  MoveL 7456 to (240.92, 51.59, 106.87) mm, rotated rx 180 ry 0 rz 180 deg; joints [-19.251, 9.742, 68.195, 59.104, 22.596, -57.051]
  Call Extruder(211.45578)
  MoveL 7457 to (240.97, 51.98, 106.87) mm, rotated rx -180 ry 0 rz 180 deg; joints [-19.29, 9.772, 68.161, 59.149, 22.631, -57.091]
  MoveL 7458 to (240.97, 51.98, 106.87) mm, rotated rx -180 ry 0 rz 180 deg; joints [-19.29, 9.772, 68.161, 59.149, 22.631, -57.091]
  Call Extruder(211.65249)
  MoveL 7459 to (241.02, 52.37, 106.87) mm, rotated rx 180 ry 0 rz 180 deg; joints [-19.329, 9.801, 68.126, 59.194, 22.666, -57.131]
  MoveL 7460 to (241.02, 52.37, 106.87) mm, rotated rx 180 ry 0 rz 180 deg; joints [-19.329, 9.801, 68.126, 59.194, 22.666, -57.131]
  Call Extruder(211.84833)
  MoveL 7461 to (241.06, 52.75, 106.87) mm, rotated rx 180 ry 0 rz 180 deg; joints [-19.368, 9.831, 68.092, 59.239, 22.702, -57.171]
  MoveL 7462 to (241.06, 52.75, 106.87) mm, rotated rx 180 ry 0 rz 180 deg; joints [-19.368, 9.831, 68.092, 59.239, 22.702, -57.171]
  Call Extruder(212.14376)
  MoveL 7463 to (241.11, 53.34, 106.87) mm, rotated rx -180 ry 0 rz 180 deg; joints [-19.428, 9.872, 68.043, 59.309, 22.756, -57.233]
  MoveL 7464 to (241.11, 53.34, 106.87) mm, rotated rx -180 ry 0 rz 180 deg; joints [-19.428, 9.872, 68.043, 59.309, 22.756, -57.233]
  Call Extruder(212.43787)
  MoveL 7465 to (241.16, 53.93, 106.87) mm, rotated rx 180 ry 0 rz 180 deg; joints [-19.488, 9.914, 67.995, 59.379, 22.81, -57.295]
  MoveL 7466 to (241.16, 53.93, 106.87) mm, rotated rx 180 ry 0 rz 180 deg; joints [-19.488, 9.914, 67.995, 59.379, 22.81, -57.295]
  Call Extruder(212.73064)
  MoveL 7467 to (241.2, 54.52, 106.87) mm, rotated rx 180 ry 0 rz 180 deg; joints [-19.548, 9.956, 67.946, 59.448, 22.864, -57.357]
  MoveL 7468 to (241.2, 54.52, 106.87) mm, rotated rx 180 ry 0 rz 180 deg; joints [-19.548, 9.956, 67.946, 59.448, 22.864, -57.357]
  Call Extruder(213.30409)
  MoveL 7469 to (241.25, 55.68, 106.87) mm, rotated rx 180 ry 0 rz 180 deg; joints [-19.668, 10.031, 67.858, 59.588, 22.971, -57.482]
  MoveL 7470 to (241.25, 55.68, 106.87) mm, rotated rx 180 ry 0 rz 180 deg; joints [-19.668, 10.031, 67.858, 59.588, 22.971, -57.482]
  Call Extruder(214.01793)
  MoveL 7471 to (241.29, 57.14, 106.87) mm, rotated rx 180 ry 0 rz 180 deg; joints [-19.819, 10.123, 67.751, 59.763, 23.106, -57.637]
  Call Extruder(256.08281)
  MoveL 7472 to (241.29, 142.86, 106.87) mm, rotated rx -180 ry 0 rz 180 deg; joints [-28.232, 16.484, 59.966, 66.424, 31.073, -63.002]
  Call Extruder(256.51124)
  MoveL 7473 to (241.27, 143.73, 106.87) mm, rotated rx 180 ry 0 rz -180 deg; joints [-28.313, 16.56, 59.868, 66.463, 31.153, -63.025]
  MoveL 7474 to (241.27, 143.73, 106.87) mm, rotated rx 180 ry 0 rz -180 deg; joints [-28.313, 16.56, 59.868, 66.463, 31.153, -63.025]
  Call Extruder(257.08469)
  MoveL 7475 to (241.22, 144.9, 106.87) mm, rotated rx 180 ry 0 rz 180 deg; joints [-28.421, 16.658, 59.742, 66.516, 31.261, -63.057]
  MoveL 7476 to (241.22, 144.9, 106.87) mm, rotated rx 180 ry 0 rz 180 deg; joints [-28.421, 16.658, 59.742, 66.516, 31.261, -63.057]
  Call Extruder(257.51903)
  MoveL 7477 to (241.18, 145.77, 106.87) mm, rotated rx -180 ry 0 rz 180 deg; joints [-28.503, 16.731, 59.649, 66.557, 31.342, -63.082]
  MoveL 7478 to (241.18, 145.77, 106.87) mm, rotated rx -180 ry 0 rz 180 deg; joints [-28.503, 16.731, 59.649, 66.557, 31.342, -63.082]
  Call Extruder(257.81314)
  MoveL 7479 to (241.13, 146.36, 106.87) mm, rotated rx 180 ry 0 rz 180 deg; joints [-28.559, 16.777, 59.59, 66.586, 31.397, -63.101]
  MoveL 7480 to (241.13, 146.36, 106.87) mm, rotated rx 180 ry 0 rz 180 deg; joints [-28.559, 16.777, 59.59, 66.586, 31.397, -63.101]
  Call Extruder(258.10858)
  MoveL 7481 to (241.09, 146.95, 106.87) mm, rotated rx 180 ry 0 rz 180 deg; joints [-28.615, 16.824, 59.53, 66.615, 31.452, -63.119]
  MoveL 7482 to (241.09, 146.95, 106.87) mm, rotated rx 180 ry 0 rz 180 deg; joints [-28.615, 16.824, 59.53, 66.615, 31.452, -63.119]
  Call Extruder(258.35483)
  MoveL 7483 to (241.04, 147.44, 106.87) mm, rotated rx -180 ry 0 rz 180 deg; joints [-28.662, 16.861, 59.482, 66.639, 31.498, -63.135]
  MoveL 7484 to (241.04, 147.44, 106.87) mm, rotated rx -180 ry 0 rz 180 deg; joints [-28.662, 16.861, 59.482, 66.639, 31.498, -63.135]
  Call Extruder(258.55154)
  MoveL 7485 to (240.99, 147.83, 106.87) mm, rotated rx -180 ry 0 rz 180 deg; joints [-28.7, 16.889, 59.446, 66.66, 31.535, -63.148]
  MoveL 7486 to (240.99, 147.83, 106.87) mm, rotated rx -180 ry 0 rz 180 deg; joints [-28.7, 16.889, 59.446, 66.66, 31.535, -63.148]
  Call Extruder(258.74911)
  MoveL 7487 to (240.95, 148.22, 106.87) mm, rotated rx 180 ry 0 rz 180 deg; joints [-28.737, 16.917, 59.41, 66.68, 31.571, -63.162]
  MoveL 7488 to (240.95, 148.22, 106.87) mm, rotated rx 180 ry 0 rz 180 deg; joints [-28.737, 16.917, 59.41, 66.68, 31.571, -63.162]
  Call Extruder(258.94755)
  MoveL 7489 to (240.9, 148.6, 106.87) mm, rotated rx 180 ry 0 rz 180 deg; joints [-28.774, 16.945, 59.374, 66.7, 31.608, -63.175]
  MoveL 7490 to (240.9, 148.6, 106.87) mm, rotated rx 180 ry 0 rz 180 deg; joints [-28.774, 16.945, 59.374, 66.7, 31.608, -63.175]
  Call Extruder(259.14686)
  MoveL 7491 to (240.86, 148.99, 106.87) mm, rotated rx 180 ry 0 rz 180 deg; joints [-28.812, 16.974, 59.338, 66.72, 31.645, -63.188]
  MoveL 7492 to (240.86, 148.99, 106.87) mm, rotated rx 180 ry 0 rz 180 deg; joints [-28.812, 16.974, 59.338, 66.72, 31.645, -63.188]
  Call Extruder(259.30569)
  MoveL 7493 to (240.81, 149.3, 106.87) mm, rotated rx 180 ry 0 rz 180 deg; joints [-28.842, 16.994, 59.311, 66.737, 31.674, -63.2]
  MoveL 7494 to (240.81, 149.3, 106.87) mm, rotated rx 180 ry 0 rz 180 deg; joints [-28.842, 16.994, 59.311, 66.737, 31.674, -63.2]
  Call Extruder(259.46525)
  MoveL 7495 to (240.76, 149.6, 106.87) mm, rotated rx -180 ry 0 rz 180 deg; joints [-28.872, 17.014, 59.285, 66.755, 31.703, -63.212]
  MoveL 7496 to (240.76, 149.6, 106.87) mm, rotated rx -180 ry 0 rz 180 deg; joints [-28.872, 17.014, 59.285, 66.755, 31.703, -63.212]
  Call Extruder(259.62554)
  MoveL 7497 to (240.71, 149.91, 106.87) mm, rotated rx 180 ry 0 rz 180 deg; joints [-28.902, 17.035, 59.259, 66.772, 31.732, -63.224]
  MoveL 7498 to (240.71, 149.91, 106.87) mm, rotated rx 180 ry 0 rz 180 deg; joints [-28.902, 17.035, 59.259, 66.772, 31.732, -63.224]
  Call Extruder(259.78655)
  MoveL 7499 to (240.66, 150.21, 106.87) mm, rotated rx -180 ry 0 rz -180 deg; joints [-28.932, 17.055, 59.233, 66.789, 31.761, -63.236]
  MoveL 7500 to (240.66, 150.21, 106.87) mm, rotated rx -180 ry 0 rz -180 deg; joints [-28.932, 17.055, 59.233, 66.789, 31.761, -63.236]
  Call Extruder(259.94830)
  MoveL 7501 to (240.61, 150.52, 106.87) mm, rotated rx 180 ry 0 rz 180 deg; joints [-28.962, 17.075, 59.207, 66.806, 31.791, -63.247]
  MoveL 7502 to (240.61, 150.52, 106.87) mm, rotated rx 180 ry 0 rz 180 deg; joints [-28.962, 17.075, 59.207, 66.806, 31.791, -63.247]
  Call Extruder(260.11077)
  MoveL 7503 to (240.57, 150.83, 106.87) mm, rotated rx -180 ry 0 rz 180 deg; joints [-28.993, 17.096, 59.18, 66.823, 31.82, -63.259]
  MoveL 7504 to (240.57, 150.83, 106.87) mm, rotated rx -180 ry 0 rz 180 deg; joints [-28.993, 17.096, 59.18, 66.823, 31.82, -63.259]
  Call Extruder(260.24469)
  MoveL 7505 to (240.52, 151.08, 106.87) mm, rotated rx 180 ry 0 rz 180 deg; joints [-29.017, 17.111, 59.161, 66.838, 31.844, -63.269]
  MoveL 7506 to (240.52, 151.08, 106.87) mm, rotated rx 180 ry 0 rz 180 deg; joints [-29.017, 17.111, 59.161, 66.838, 31.844, -63.269]
  Call Extruder(260.37923)
  MoveL 7507 to (240.47, 151.32, 106.87) mm, rotated rx -180 ry 0 rz 180 deg; joints [-29.043, 17.126, 59.142, 66.853, 31.868, -63.28]
  MoveL 7508 to (240.47, 151.32, 106.87) mm, rotated rx -180 ry 0 rz 180 deg; joints [-29.043, 17.126, 59.142, 66.853, 31.868, -63.28]
  Call Extruder(260.51438)
  MoveL 7509 to (240.42, 151.57, 106.87) mm, rotated rx 180 ry 0 rz 180 deg; joints [-29.067, 17.141, 59.122, 66.868, 31.892, -63.29]
  MoveL 7510 to (240.42, 151.57, 106.87) mm, rotated rx 180 ry 0 rz 180 deg; joints [-29.067, 17.141, 59.122, 66.868, 31.892, -63.29]
  Call Extruder(260.65014)
  MoveL 7511 to (240.37, 151.82, 106.87) mm, rotated rx -180 ry 0 rz 180 deg; joints [-29.092, 17.156, 59.103, 66.882, 31.916, -63.301]
  MoveL 7512 to (240.37, 151.82, 106.87) mm, rotated rx -180 ry 0 rz 180 deg; joints [-29.092, 17.156, 59.103, 66.882, 31.916, -63.301]
  Call Extruder(260.78650)
  MoveL 7513 to (240.32, 152.07, 106.87) mm, rotated rx 180 ry 0 rz 180 deg; joints [-29.117, 17.171, 59.083, 66.897, 31.94, -63.311]
  MoveL 7514 to (240.32, 152.07, 106.87) mm, rotated rx 180 ry 0 rz 180 deg; joints [-29.117, 17.171, 59.083, 66.897, 31.94, -63.311]
  Call Extruder(260.92348)
  MoveL 7515 to (240.27, 152.32, 106.87) mm, rotated rx -180 ry 0 rz 180 deg; joints [-29.142, 17.186, 59.064, 66.912, 31.964, -63.321]
  MoveL 7516 to (240.27, 152.32, 106.87) mm, rotated rx -180 ry 0 rz 180 deg; joints [-29.142, 17.186, 59.064, 66.912, 31.964, -63.321]
  Call Extruder(261.06107)
  MoveL 7517 to (240.22, 152.57, 106.87) mm, rotated rx -180 ry 0 rz 180 deg; joints [-29.167, 17.201, 59.044, 66.926, 31.988, -63.332]
  MoveL 7518 to (240.22, 152.57, 106.87) mm, rotated rx -180 ry 0 rz 180 deg; joints [-29.167, 17.201, 59.044, 66.926, 31.988, -63.332]
  Call Extruder(261.17477)
  MoveL 7519 to (240.17, 152.77, 106.87) mm, rotated rx 180 ry 0 rz 180 deg; joints [-29.188, 17.213, 59.029, 66.939, 32.008, -63.341]
  MoveL 7520 to (240.17, 152.77, 106.87) mm, rotated rx 180 ry 0 rz 180 deg; joints [-29.188, 17.213, 59.029, 66.939, 32.008, -63.341]
  Call Extruder(261.28892)
  MoveL 7521 to (240.13, 152.98, 106.87) mm, rotated rx 180 ry 0 rz 180 deg; joints [-29.209, 17.225, 59.014, 66.951, 32.027, -63.35]
  MoveL 7522 to (240.13, 152.98, 106.87) mm, rotated rx 180 ry 0 rz 180 deg; joints [-29.209, 17.225, 59.014, 66.951, 32.027, -63.35]
  Call Extruder(261.40352)
  MoveL 7523 to (240.08, 153.18, 106.87) mm, rotated rx 180 ry 0 rz 180 deg; joints [-29.229, 17.237, 58.999, 66.964, 32.047, -63.358]
  MoveL 7524 to (240.08, 153.18, 106.87) mm, rotated rx 180 ry 0 rz 180 deg; joints [-29.229, 17.237, 58.999, 66.964, 32.047, -63.358]
  Call Extruder(261.51858)
  MoveL 7525 to (240.04, 153.39, 106.87) mm, rotated rx 180 ry 0 rz 180 deg; joints [-29.25, 17.248, 58.983, 66.976, 32.067, -63.367]
  MoveL 7526 to (240.04, 153.39, 106.87) mm, rotated rx 180 ry 0 rz 180 deg; joints [-29.25, 17.248, 58.983, 66.976, 32.067, -63.367]
  Call Extruder(261.64080)
  MoveL 7527 to (239.98, 153.6, 106.87) mm, rotated rx 180 ry 0 rz 180 deg; joints [-29.272, 17.259, 58.97, 66.99, 32.088, -63.378]
  MoveL 7528 to (239.98, 153.6, 106.87) mm, rotated rx 180 ry 0 rz 180 deg; joints [-29.272, 17.259, 58.97, 66.99, 32.088, -63.378]
  Call Extruder(261.77046)
  MoveL 7529 to (239.92, 153.82, 106.87) mm, rotated rx -180 ry 0 rz 180 deg; joints [-29.296, 17.269, 58.957, 67.006, 32.11, -63.389]
  MoveL 7530 to (239.92, 153.82, 106.87) mm, rotated rx -180 ry 0 rz 180 deg; joints [-29.296, 17.269, 58.957, 67.006, 32.11, -63.389]
  Call Extruder(261.90069)
  MoveL 7531 to (239.85, 154.05, 106.87) mm, rotated rx 180 ry 0 rz 180 deg; joints [-29.319, 17.279, 58.944, 67.021, 32.132, -63.401]
  MoveL 7532 to (239.85, 154.05, 106.87) mm, rotated rx 180 ry 0 rz 180 deg; joints [-29.319, 17.279, 58.944, 67.021, 32.132, -63.401]
  Call Extruder(262.03148)
  MoveL 7533 to (239.78, 154.27, 106.87) mm, rotated rx 180 ry 0 rz 180 deg; joints [-29.343, 17.289, 58.932, 67.037, 32.155, -63.413]
  MoveL 7534 to (239.78, 154.27, 106.87) mm, rotated rx 180 ry 0 rz 180 deg; joints [-29.343, 17.289, 58.932, 67.037, 32.155, -63.413]
  Call Extruder(262.16284)
  MoveL 7535 to (239.71, 154.5, 106.87) mm, rotated rx 180 ry 0 rz -180 deg; joints [-29.366, 17.299, 58.919, 67.053, 32.177, -63.425]
  MoveL 7536 to (239.71, 154.5, 106.87) mm, rotated rx 180 ry 0 rz -180 deg; joints [-29.366, 17.299, 58.919, 67.053, 32.177, -63.425]
  Call Extruder(262.27474)
  MoveL 7537 to (239.65, 154.68, 106.87) mm, rotated rx 180 ry 0 rz 180 deg; joints [-29.386, 17.306, 58.909, 67.066, 32.195, -63.435]
  MoveL 7538 to (239.65, 154.68, 106.87) mm, rotated rx 180 ry 0 rz 180 deg; joints [-29.386, 17.306, 58.909, 67.066, 32.195, -63.435]
  Call Extruder(262.38708)
  MoveL 7539 to (239.59, 154.87, 106.87) mm, rotated rx 180 ry 0 rz -180 deg; joints [-29.406, 17.314, 58.899, 67.08, 32.214, -63.446]
  MoveL 7540 to (239.59, 154.87, 106.87) mm, rotated rx 180 ry 0 rz -180 deg; joints [-29.406, 17.314, 58.899, 67.08, 32.214, -63.446]
  Call Extruder(262.49987)
  MoveL 7541 to (239.53, 155.06, 106.87) mm, rotated rx 180 ry 0 rz 180 deg; joints [-29.426, 17.321, 58.889, 67.093, 32.233, -63.456]
  MoveL 7542 to (239.53, 155.06, 106.87) mm, rotated rx 180 ry 0 rz 180 deg; joints [-29.426, 17.321, 58.889, 67.093, 32.233, -63.456]
  Call Extruder(262.61311)
  MoveL 7543 to (239.47, 155.25, 106.87) mm, rotated rx 180 ry 0 rz 180 deg; joints [-29.446, 17.329, 58.879, 67.107, 32.252, -63.466]
  MoveL 7544 to (239.47, 155.25, 106.87) mm, rotated rx 180 ry 0 rz 180 deg; joints [-29.446, 17.329, 58.879, 67.107, 32.252, -63.466]
  Call Extruder(262.72679)
  MoveL 7545 to (239.41, 155.44, 106.87) mm, rotated rx 180 ry 0 rz 180 deg; joints [-29.466, 17.337, 58.87, 67.12, 32.271, -63.477]
  MoveL 7546 to (239.41, 155.44, 106.87) mm, rotated rx 180 ry 0 rz 180 deg; joints [-29.466, 17.337, 58.87, 67.12, 32.271, -63.477]
  Call Extruder(262.90875)
  MoveL 7547 to (239.29, 155.73, 106.87) mm, rotated rx -180 ry 0 rz 180 deg; joints [-29.499, 17.344, 58.86, 67.144, 32.3, -63.496]
  MoveL 7548 to (239.29, 155.73, 106.87) mm, rotated rx -180 ry 0 rz 180 deg; joints [-29.499, 17.344, 58.86, 67.144, 32.3, -63.496]
  Call Extruder(263.09146)
  MoveL 7549 to (239.17, 156.02, 106.87) mm, rotated rx 180 ry 0 rz 180 deg; joints [-29.531, 17.352, 58.85, 67.168, 32.33, -63.515]
  MoveL 7550 to (239.17, 156.02, 106.87) mm, rotated rx 180 ry 0 rz 180 deg; joints [-29.531, 17.352, 58.85, 67.168, 32.33, -63.515]
  Call Extruder(263.26189)
  MoveL 7551 to (239.05, 156.29, 106.87) mm, rotated rx 180 ry 0 rz 180 deg; joints [-29.561, 17.358, 58.842, 67.19, 32.358, -63.533]
  MoveL 7552 to (239.05, 156.29, 106.87) mm, rotated rx 180 ry 0 rz 180 deg; joints [-29.561, 17.358, 58.842, 67.19, 32.358, -63.533]
  Call Extruder(263.41990)
  MoveL 7553 to (238.94, 156.54, 106.87) mm, rotated rx 180 ry 0 rz 180 deg; joints [-29.589, 17.364, 58.834, 67.211, 32.383, -63.549]
  MoveL 7554 to (238.94, 156.54, 106.87) mm, rotated rx 180 ry 0 rz 180 deg; joints [-29.589, 17.364, 58.834, 67.211, 32.383, -63.549]
  Call Extruder(263.57851)
  MoveL 7555 to (238.84, 156.79, 106.87) mm, rotated rx 180 ry 0 rz 180 deg; joints [-29.617, 17.37, 58.827, 67.231, 32.409, -63.566]
  MoveL 7556 to (238.84, 156.79, 106.87) mm, rotated rx 180 ry 0 rz 180 deg; joints [-29.617, 17.37, 58.827, 67.231, 32.409, -63.566]
  Call Extruder(263.78468)
  MoveL 7557 to (238.66, 157.09, 106.87) mm, rotated rx 180 ry 0 rz 180 deg; joints [-29.653, 17.37, 58.827, 67.262, 32.441, -63.591]
  MoveL 7558 to (238.66, 157.09, 106.87) mm, rotated rx 180 ry 0 rz 180 deg; joints [-29.653, 17.37, 58.827, 67.262, 32.441, -63.591]
  Call Extruder(263.99163)
  MoveL 7559 to (238.49, 157.4, 106.87) mm, rotated rx 180 ry 0 rz 180 deg; joints [-29.689, 17.369, 58.828, 67.292, 32.474, -63.617]
  MoveL 7560 to (238.49, 157.4, 106.87) mm, rotated rx 180 ry 0 rz 180 deg; joints [-29.689, 17.369, 58.828, 67.292, 32.474, -63.617]
  Call Extruder(264.19935)
  MoveL 7561 to (238.31, 157.7, 106.87) mm, rotated rx 180 ry 0 rz -180 deg; joints [-29.725, 17.369, 58.828, 67.322, 32.506, -63.642]
  MoveL 7562 to (238.31, 157.7, 106.87) mm, rotated rx 180 ry 0 rz -180 deg; joints [-29.725, 17.369, 58.828, 67.322, 32.506, -63.642]
  Call Extruder(264.40786)
  MoveL 7563 to (238.13, 158.01, 106.87) mm, rotated rx 180 ry 0 rz 180 deg; joints [-29.761, 17.368, 58.828, 67.352, 32.538, -63.668]
  MoveL 7564 to (238.13, 158.01, 106.87) mm, rotated rx 180 ry 0 rz 180 deg; joints [-29.761, 17.368, 58.828, 67.352, 32.538, -63.668]
  Call Extruder(264.58740)
  MoveL 7565 to (237.96, 158.25, 106.87) mm, rotated rx 180 ry 0 rz 180 deg; joints [-29.792, 17.362, 58.836, 67.38, 32.566, -63.692]
  MoveL 7566 to (237.96, 158.25, 106.87) mm, rotated rx 180 ry 0 rz 180 deg; joints [-29.792, 17.362, 58.836, 67.38, 32.566, -63.692]
  Call Extruder(264.92080)
  MoveL 7567 to (237.63, 158.7, 106.87) mm, rotated rx 180 ry 0 rz 180 deg; joints [-29.849, 17.351, 58.851, 67.432, 32.615, -63.738]
  MoveL 7568 to (237.63, 158.7, 106.87) mm, rotated rx 180 ry 0 rz 180 deg; joints [-29.849, 17.351, 58.851, 67.432, 32.615, -63.738]
  Call Extruder(265.25540)
  MoveL 7569 to (237.3, 159.15, 106.87) mm, rotated rx -180 ry 0 rz 180 deg; joints [-29.907, 17.339, 58.866, 67.484, 32.666, -63.783]
  Call Extruder(266.08335)
  MoveL 7570 to (236.39, 160.19, 106.87) mm, rotated rx 180 ry 0 rz 180 deg; joints [-30.046, 17.286, 58.935, 67.62, 32.785, -63.905]
  Call Extruder(266.91129)
  MoveL 7571 to (235.35, 161.1, 106.87) mm, rotated rx 180 ry 0 rz 180 deg; joints [-30.182, 17.201, 59.045, 67.765, 32.897, -64.039]
  Call Extruder(267.07860)
  MoveL 7572 to (235.13, 161.27, 106.87) mm, rotated rx 180 ry 0 rz 180 deg; joints [-30.208, 17.179, 59.073, 67.795, 32.918, -64.068]
  MoveL 7573 to (235.13, 161.27, 106.87) mm, rotated rx 180 ry 0 rz 180 deg; joints [-30.208, 17.179, 59.073, 67.795, 32.918, -64.068]
  Call Extruder(267.41202)
  MoveL 7574 to (234.68, 161.6, 106.87) mm, rotated rx 180 ry 0 rz 180 deg; joints [-30.261, 17.136, 59.129, 67.855, 32.961, -64.125]
  MoveL 7575 to (234.68, 161.6, 106.87) mm, rotated rx 180 ry 0 rz 180 deg; joints [-30.261, 17.136, 59.129, 67.855, 32.961, -64.125]
  Call Extruder(267.74426)
  MoveL 7576 to (234.23, 161.92, 106.87) mm, rotated rx 180 ry 0 rz 180 deg; joints [-30.314, 17.092, 59.185, 67.916, 33.004, -64.182]
  MoveL 7577 to (234.23, 161.92, 106.87) mm, rotated rx 180 ry 0 rz 180 deg; joints [-30.314, 17.092, 59.185, 67.916, 33.004, -64.182]
  Call Extruder(267.86192)
  MoveL 7578 to (234.05, 162.02, 106.87) mm, rotated rx 180 ry 0 rz -180 deg; joints [-30.331, 17.073, 59.209, 67.938, 33.018, -64.203]
  MoveL 7579 to (234.05, 162.02, 106.87) mm, rotated rx 180 ry 0 rz -180 deg; joints [-30.331, 17.073, 59.209, 67.938, 33.018, -64.203]
  Call Extruder(268.06964)
  MoveL 7580 to (233.75, 162.2, 106.87) mm, rotated rx 180 ry 0 rz 180 deg; joints [-30.363, 17.04, 59.253, 67.977, 33.043, -64.24]
  MoveL 7581 to (233.75, 162.2, 106.87) mm, rotated rx 180 ry 0 rz 180 deg; joints [-30.363, 17.04, 59.253, 67.977, 33.043, -64.24]
  Call Extruder(268.27659)
  MoveL 7582 to (233.45, 162.37, 106.87) mm, rotated rx 180 ry 0 rz 180 deg; joints [-30.394, 17.006, 59.296, 68.015, 33.067, -64.278]
  MoveL 7583 to (233.45, 162.37, 106.87) mm, rotated rx 180 ry 0 rz 180 deg; joints [-30.394, 17.006, 59.296, 68.015, 33.067, -64.278]
  Call Extruder(268.48276)
  MoveL 7584 to (233.14, 162.55, 106.87) mm, rotated rx -180 ry 0 rz -180 deg; joints [-30.426, 16.973, 59.339, 68.054, 33.092, -64.315]
  MoveL 7585 to (233.14, 162.55, 106.87) mm, rotated rx -180 ry 0 rz -180 deg; joints [-30.426, 16.973, 59.339, 68.054, 33.092, -64.315]
  Call Extruder(268.66443)
  MoveL 7586 to (232.87, 162.69, 106.87) mm, rotated rx 180 ry 0 rz 180 deg; joints [-30.453, 16.94, 59.38, 68.089, 33.113, -64.349]
  MoveL 7587 to (232.87, 162.69, 106.87) mm, rotated rx 180 ry 0 rz 180 deg; joints [-30.453, 16.94, 59.38, 68.089, 33.113, -64.349]
  Call Extruder(268.82240)
  MoveL 7588 to (232.62, 162.8, 106.87) mm, rotated rx 180 ry 0 rz 180 deg; joints [-30.476, 16.909, 59.42, 68.119, 33.13, -64.379]
  MoveL 7589 to (232.62, 162.8, 106.87) mm, rotated rx 180 ry 0 rz 180 deg; joints [-30.476, 16.909, 59.42, 68.119, 33.13, -64.379]
  Call Extruder(268.97977)
  MoveL 7590 to (232.37, 162.91, 106.87) mm, rotated rx 180 ry 0 rz 180 deg; joints [-30.498, 16.878, 59.46, 68.15, 33.147, -64.409]
  MoveL 7591 to (232.37, 162.91, 106.87) mm, rotated rx 180 ry 0 rz 180 deg; joints [-30.498, 16.878, 59.46, 68.15, 33.147, -64.409]
  Call Extruder(269.16252)
  MoveL 7592 to (232.08, 163.03, 106.87) mm, rotated rx 180 ry 0 rz 180 deg; joints [-30.524, 16.842, 59.507, 68.185, 33.167, -64.444]
  MoveL 7593 to (232.08, 163.03, 106.87) mm, rotated rx 180 ry 0 rz 180 deg; joints [-30.524, 16.842, 59.507, 68.185, 33.167, -64.444]
  Call Extruder(269.34450)
  MoveL 7594 to (231.78, 163.15, 106.87) mm, rotated rx 180 ry 0 rz -180 deg; joints [-30.551, 16.805, 59.554, 68.22, 33.187, -64.479]
  MoveL 7595 to (231.78, 163.15, 106.87) mm, rotated rx 180 ry 0 rz -180 deg; joints [-30.551, 16.805, 59.554, 68.22, 33.187, -64.479]
  Call Extruder(269.49184)
  MoveL 7596 to (231.54, 163.24, 106.87) mm, rotated rx 180 ry 0 rz 180 deg; joints [-30.571, 16.774, 59.594, 68.249, 33.202, -64.507]
  MoveL 7597 to (231.54, 163.24, 106.87) mm, rotated rx 180 ry 0 rz 180 deg; joints [-30.571, 16.774, 59.594, 68.249, 33.202, -64.507]
  Call Extruder(269.60506)
  MoveL 7598 to (231.35, 163.3, 106.87) mm, rotated rx 180 ry 0 rz 180 deg; joints [-30.587, 16.749, 59.626, 68.271, 33.214, -64.529]
  MoveL 7599 to (231.35, 163.3, 106.87) mm, rotated rx 180 ry 0 rz 180 deg; joints [-30.587, 16.749, 59.626, 68.271, 33.214, -64.529]
  Call Extruder(269.71784)
  MoveL 7600 to (231.17, 163.36, 106.87) mm, rotated rx 180 ry 0 rz 180 deg; joints [-30.602, 16.724, 59.658, 68.294, 33.225, -64.552]
  MoveL 7601 to (231.17, 163.36, 106.87) mm, rotated rx 180 ry 0 rz 180 deg; joints [-30.602, 16.724, 59.658, 68.294, 33.225, -64.552]
  Call Extruder(269.83017)
  MoveL 7602 to (230.98, 163.42, 106.87) mm, rotated rx 180 ry 0 rz 180 deg; joints [-30.618, 16.699, 59.691, 68.316, 33.236, -64.574]
  MoveL 7603 to (230.98, 163.42, 106.87) mm, rotated rx 180 ry 0 rz 180 deg; joints [-30.618, 16.699, 59.691, 68.316, 33.236, -64.574]
  Call Extruder(269.94206)
  MoveL 7604 to (230.79, 163.48, 106.87) mm, rotated rx 180 ry 0 rz 180 deg; joints [-30.633, 16.673, 59.723, 68.338, 33.248, -64.596]
  MoveL 7605 to (230.79, 163.48, 106.87) mm, rotated rx 180 ry 0 rz 180 deg; joints [-30.633, 16.673, 59.723, 68.338, 33.248, -64.596]
  Call Extruder(270.06346)
  MoveL 7606 to (230.58, 163.55, 106.87) mm, rotated rx -180 ry 0 rz 180 deg; joints [-30.65, 16.646, 59.758, 68.362, 33.26, -64.62]
  MoveL 7607 to (230.58, 163.55, 106.87) mm, rotated rx -180 ry 0 rz 180 deg; joints [-30.65, 16.646, 59.758, 68.362, 33.26, -64.62]
  Call Extruder(270.19428)
  MoveL 7608 to (230.36, 163.62, 106.87) mm, rotated rx 180 ry 0 rz 180 deg; joints [-30.668, 16.615, 59.797, 68.388, 33.273, -64.646]
  MoveL 7609 to (230.36, 163.62, 106.87) mm, rotated rx 180 ry 0 rz 180 deg; joints [-30.668, 16.615, 59.797, 68.388, 33.273, -64.646]
  Call Extruder(270.32452)
  MoveL 7610 to (230.14, 163.68, 106.87) mm, rotated rx 180 ry 0 rz 180 deg; joints [-30.685, 16.585, 59.836, 68.414, 33.286, -64.672]
  MoveL 7611 to (230.14, 163.68, 106.87) mm, rotated rx 180 ry 0 rz 180 deg; joints [-30.685, 16.585, 59.836, 68.414, 33.286, -64.672]
  Call Extruder(270.45421)
  MoveL 7612 to (229.91, 163.75, 106.87) mm, rotated rx 180 ry 0 rz 180 deg; joints [-30.703, 16.555, 59.875, 68.44, 33.299, -64.698]
  MoveL 7613 to (229.91, 163.75, 106.87) mm, rotated rx 180 ry 0 rz 180 deg; joints [-30.703, 16.555, 59.875, 68.44, 33.299, -64.698]
  Call Extruder(270.58333)
  MoveL 7614 to (229.69, 163.82, 106.87) mm, rotated rx 180 ry 0 rz 180 deg; joints [-30.721, 16.525, 59.913, 68.466, 33.312, -64.724]
  MoveL 7615 to (229.69, 163.82, 106.87) mm, rotated rx 180 ry 0 rz 180 deg; joints [-30.721, 16.525, 59.913, 68.466, 33.312, -64.724]
  Call Extruder(270.69840)
  MoveL 7616 to (229.48, 163.86, 106.87) mm, rotated rx 180 ry 0 rz 180 deg; joints [-30.736, 16.495, 59.951, 68.489, 33.322, -64.747]
  MoveL 7617 to (229.48, 163.86, 106.87) mm, rotated rx 180 ry 0 rz 180 deg; joints [-30.736, 16.495, 59.951, 68.489, 33.322, -64.747]
  Call Extruder(270.81302)
  MoveL 7618 to (229.28, 163.91, 106.87) mm, rotated rx 180 ry 0 rz 180 deg; joints [-30.751, 16.466, 59.988, 68.512, 33.333, -64.771]
  MoveL 7619 to (229.28, 163.91, 106.87) mm, rotated rx 180 ry 0 rz 180 deg; joints [-30.751, 16.466, 59.988, 68.512, 33.333, -64.771]
  Call Extruder(270.92719)
  MoveL 7620 to (229.08, 163.95, 106.87) mm, rotated rx -180 ry 0 rz -180 deg; joints [-30.766, 16.437, 60.025, 68.535, 33.343, -64.794]
  MoveL 7621 to (229.08, 163.95, 106.87) mm, rotated rx -180 ry 0 rz -180 deg; joints [-30.766, 16.437, 60.025, 68.535, 33.343, -64.794]
  Call Extruder(271.04091)
  MoveL 7622 to (228.87, 164, 106.87) mm, rotated rx 180 ry 0 rz 180 deg; joints [-30.781, 16.408, 60.063, 68.558, 33.354, -64.817]
  MoveL 7623 to (228.87, 164, 106.87) mm, rotated rx 180 ry 0 rz 180 deg; joints [-30.781, 16.408, 60.063, 68.558, 33.354, -64.817]
  Call Extruder(271.16633)
  MoveL 7624 to (228.64, 164.04, 106.87) mm, rotated rx 180 ry 0 rz -180 deg; joints [-30.797, 16.375, 60.104, 68.583, 33.365, -64.843]
  MoveL 7625 to (228.64, 164.04, 106.87) mm, rotated rx 180 ry 0 rz -180 deg; joints [-30.797, 16.375, 60.104, 68.583, 33.365, -64.843]
  Call Extruder(271.30331)
  MoveL 7626 to (228.4, 164.09, 106.87) mm, rotated rx -180 ry 0 rz 180 deg; joints [-30.815, 16.339, 60.15, 68.611, 33.378, -64.871]
  MoveL 7627 to (228.4, 164.09, 106.87) mm, rotated rx -180 ry 0 rz 180 deg; joints [-30.815, 16.339, 60.15, 68.611, 33.378, -64.871]
  Call Extruder(271.43968)
  MoveL 7628 to (228.15, 164.14, 106.87) mm, rotated rx 180 ry 0 rz 180 deg; joints [-30.832, 16.303, 60.196, 68.638, 33.39, -64.9]
  MoveL 7629 to (228.15, 164.14, 106.87) mm, rotated rx 180 ry 0 rz 180 deg; joints [-30.832, 16.303, 60.196, 68.638, 33.39, -64.9]
  Call Extruder(271.57543)
  MoveL 7630 to (227.9, 164.19, 106.87) mm, rotated rx -180 ry 0 rz 180 deg; joints [-30.85, 16.267, 60.242, 68.666, 33.403, -64.928]
  MoveL 7631 to (227.9, 164.19, 106.87) mm, rotated rx -180 ry 0 rz 180 deg; joints [-30.85, 16.267, 60.242, 68.666, 33.403, -64.928]
  Call Extruder(271.71058)
  MoveL 7632 to (227.65, 164.24, 106.87) mm, rotated rx 180 ry 0 rz 180 deg; joints [-30.868, 16.231, 60.288, 68.694, 33.415, -64.956]
  MoveL 7633 to (227.65, 164.24, 106.87) mm, rotated rx 180 ry 0 rz 180 deg; joints [-30.868, 16.231, 60.288, 68.694, 33.415, -64.956]
  Call Extruder(271.84512)
  MoveL 7634 to (227.4, 164.29, 106.87) mm, rotated rx 180 ry 0 rz 180 deg; joints [-30.886, 16.195, 60.333, 68.721, 33.428, -64.984]
  MoveL 7635 to (227.4, 164.29, 106.87) mm, rotated rx 180 ry 0 rz 180 deg; joints [-30.886, 16.195, 60.333, 68.721, 33.428, -64.984]
  Call Extruder(271.97904)
  MoveL 7636 to (227.15, 164.34, 106.87) mm, rotated rx -180 ry 0 rz 180 deg; joints [-30.903, 16.16, 60.379, 68.748, 33.44, -65.012]
  MoveL 7637 to (227.15, 164.34, 106.87) mm, rotated rx -180 ry 0 rz 180 deg; joints [-30.903, 16.16, 60.379, 68.748, 33.44, -65.012]
  Call Extruder(272.12691)
  MoveL 7638 to (226.87, 164.39, 106.87) mm, rotated rx -180 ry 0 rz 180 deg; joints [-30.923, 16.119, 60.431, 68.779, 33.454, -65.042]
  MoveL 7639 to (226.87, 164.39, 106.87) mm, rotated rx -180 ry 0 rz 180 deg; joints [-30.923, 16.119, 60.431, 68.779, 33.454, -65.042]
  Call Extruder(272.28865)
  MoveL 7640 to (226.57, 164.44, 106.87) mm, rotated rx 180 ry 0 rz 180 deg; joints [-30.943, 16.074, 60.488, 68.812, 33.468, -65.076]
  MoveL 7641 to (226.57, 164.44, 106.87) mm, rotated rx 180 ry 0 rz 180 deg; joints [-30.943, 16.074, 60.488, 68.812, 33.468, -65.076]
  Call Extruder(272.44966)
  MoveL 7642 to (226.26, 164.49, 106.87) mm, rotated rx 180 ry 0 rz 180 deg; joints [-30.964, 16.029, 60.545, 68.845, 33.482, -65.11]
  MoveL 7643 to (226.26, 164.49, 106.87) mm, rotated rx 180 ry 0 rz 180 deg; joints [-30.964, 16.029, 60.545, 68.845, 33.482, -65.11]
  Call Extruder(272.60995)
  MoveL 7644 to (225.95, 164.53, 106.87) mm, rotated rx 180 ry 0 rz 180 deg; joints [-30.985, 15.984, 60.602, 68.878, 33.497, -65.144]
  MoveL 7645 to (225.95, 164.53, 106.87) mm, rotated rx 180 ry 0 rz 180 deg; joints [-30.985, 15.984, 60.602, 68.878, 33.497, -65.144]
  Call Extruder(272.76951)
  MoveL 7646 to (225.65, 164.58, 106.87) mm, rotated rx 180 ry 0 rz 180 deg; joints [-31.006, 15.939, 60.659, 68.911, 33.511, -65.178]
  MoveL 7647 to (225.65, 164.58, 106.87) mm, rotated rx 180 ry 0 rz 180 deg; joints [-31.006, 15.939, 60.659, 68.911, 33.511, -65.178]
  Call Extruder(272.92834)
  MoveL 7648 to (225.34, 164.63, 106.87) mm, rotated rx 180 ry 0 rz 180 deg; joints [-31.027, 15.894, 60.716, 68.943, 33.526, -65.211]
  MoveL 7649 to (225.34, 164.63, 106.87) mm, rotated rx 180 ry 0 rz 180 deg; joints [-31.027, 15.894, 60.716, 68.943, 33.526, -65.211]
  Call Extruder(273.10701)
  MoveL 7650 to (225, 164.68, 106.87) mm, rotated rx 180 ry 0 rz -180 deg; joints [-31.049, 15.842, 60.782, 68.98, 33.542, -65.249]
  MoveL 7651 to (225, 164.68, 106.87) mm, rotated rx 180 ry 0 rz -180 deg; joints [-31.049, 15.842, 60.782, 68.98, 33.542, -65.249]
  Call Extruder(273.30545)
  MoveL 7652 to (224.61, 164.72, 106.87) mm, rotated rx -180 ry 0 rz 180 deg; joints [-31.074, 15.784, 60.856, 69.021, 33.559, -65.291]
  MoveL 7653 to (224.61, 164.72, 106.87) mm, rotated rx -180 ry 0 rz 180 deg; joints [-31.074, 15.784, 60.856, 69.021, 33.559, -65.291]
  Call Extruder(273.50302)
  MoveL 7654 to (224.22, 164.77, 106.87) mm, rotated rx -180 ry 0 rz 180 deg; joints [-31.1, 15.726, 60.929, 69.062, 33.576, -65.333]
  MoveL 7655 to (224.22, 164.77, 106.87) mm, rotated rx -180 ry 0 rz 180 deg; joints [-31.1, 15.726, 60.929, 69.062, 33.576, -65.333]
  Call Extruder(273.69973)
  MoveL 7656 to (223.84, 164.82, 106.87) mm, rotated rx -180 ry 0 rz -180 deg; joints [-31.125, 15.668, 61.003, 69.102, 33.594, -65.375]
  MoveL 7657 to (223.84, 164.82, 106.87) mm, rotated rx -180 ry 0 rz -180 deg; joints [-31.125, 15.668, 61.003, 69.102, 33.594, -65.375]
  Call Extruder(273.89557)
  MoveL 7658 to (223.45, 164.86, 106.87) mm, rotated rx -180 ry 0 rz 180 deg; joints [-31.15, 15.61, 61.076, 69.143, 33.611, -65.416]
  MoveL 7659 to (223.45, 164.86, 106.87) mm, rotated rx -180 ry 0 rz 180 deg; joints [-31.15, 15.61, 61.076, 69.143, 33.611, -65.416]
  Call Extruder(274.19092)
  MoveL 7660 to (222.86, 164.91, 106.87) mm, rotated rx 180 ry 0 rz 180 deg; joints [-31.186, 15.519, 61.19, 69.203, 33.635, -65.479]
  MoveL 7661 to (222.86, 164.91, 106.87) mm, rotated rx 180 ry 0 rz 180 deg; joints [-31.186, 15.519, 61.19, 69.203, 33.635, -65.479]
  Call Extruder(274.48494)
  MoveL 7662 to (222.27, 164.96, 106.87) mm, rotated rx -180 ry 0 rz 180 deg; joints [-31.222, 15.429, 61.304, 69.263, 33.66, -65.541]
  MoveL 7663 to (222.27, 164.96, 106.87) mm, rotated rx -180 ry 0 rz 180 deg; joints [-31.222, 15.429, 61.304, 69.263, 33.66, -65.541]
  Call Extruder(274.77764)
  MoveL 7664 to (221.68, 165, 106.87) mm, rotated rx 180 ry 0 rz 180 deg; joints [-31.258, 15.339, 61.418, 69.323, 33.685, -65.603]
  MoveL 7665 to (221.68, 165, 106.87) mm, rotated rx 180 ry 0 rz 180 deg; joints [-31.258, 15.339, 61.418, 69.323, 33.685, -65.603]
  Call Extruder(275.35108)
  MoveL 7666 to (220.52, 165.05, 106.87) mm, rotated rx -180 ry 0 rz 180 deg; joints [-31.326, 15.157, 61.646, 69.439, 33.73, -65.724]
  MoveL 7667 to (220.52, 165.05, 106.87) mm, rotated rx -180 ry 0 rz 180 deg; joints [-31.326, 15.157, 61.646, 69.439, 33.73, -65.724]
  Call Extruder(276.06510)
  MoveL 7668 to (219.06, 165.09, 106.87) mm, rotated rx -180 ry 0 rz 180 deg; joints [-31.409, 14.929, 61.932, 69.581, 33.786, -65.872]
  Call Extruder(392.91185)
  MoveL 7669 to (-19.06, 165.09, 106.87) mm, rotated rx 180 ry 0 rz 180 deg; joints [-51.475, -13.949, 91.048, 79.921, 52.618, -73.682]
  Call Extruder(393.34045)
  MoveL 7670 to (-19.94, 165.07, 106.87) mm, rotated rx -180 ry 0 rz 180 deg; joints [-51.582, -14.03, 91.11, 79.944, 52.723, -73.681]
  MoveL 7671 to (-19.94, 165.07, 106.87) mm, rotated rx -180 ry 0 rz 180 deg; joints [-51.582, -14.03, 91.11, 79.944, 52.723, -73.681]
  Call Extruder(393.91390)
  MoveL 7672 to (-21.1, 165.03, 106.87) mm, rotated rx 180 ry 0 rz 180 deg; joints [-51.722, -14.139, 91.193, 79.975, 52.863, -73.679]
  MoveL 7673 to (-21.1, 165.03, 106.87) mm, rotated rx 180 ry 0 rz 180 deg; joints [-51.722, -14.139, 91.193, 79.975, 52.863, -73.679]
  Call Extruder(394.34820)
  MoveL 7674 to (-21.97, 164.98, 106.87) mm, rotated rx 180 ry 0 rz 180 deg; joints [-51.827, -14.223, 91.257, 79.997, 52.967, -73.677]
  MoveL 7675 to (-21.97, 164.98, 106.87) mm, rotated rx 180 ry 0 rz 180 deg; joints [-51.827, -14.223, 91.257, 79.997, 52.967, -73.677]
  Call Extruder(394.64223)
  MoveL 7676 to (-22.56, 164.93, 106.87) mm, rotated rx 180 ry 0 rz 180 deg; joints [-51.897, -14.281, 91.301, 80.011, 53.036, -73.674]
  MoveL 7677 to (-22.56, 164.93, 106.87) mm, rotated rx 180 ry 0 rz 180 deg; joints [-51.897, -14.281, 91.301, 80.011, 53.036, -73.674]
  Call Extruder(394.93759)
  MoveL 7678 to (-23.15, 164.89, 106.87) mm, rotated rx 180 ry 0 rz -180 deg; joints [-51.966, -14.338, 91.345, 80.025, 53.105, -73.672]
  MoveL 7679 to (-23.15, 164.89, 106.87) mm, rotated rx 180 ry 0 rz -180 deg; joints [-51.966, -14.338, 91.345, 80.025, 53.105, -73.672]
  Call Extruder(395.18380)
  MoveL 7680 to (-23.64, 164.84, 106.87) mm, rotated rx -180 ry 0 rz 180 deg; joints [-52.023, -14.387, 91.382, 80.036, 53.161, -73.669]
  MoveL 7681 to (-23.64, 164.84, 106.87) mm, rotated rx -180 ry 0 rz 180 deg; joints [-52.023, -14.387, 91.382, 80.036, 53.161, -73.669]
  Call Extruder(395.38051)
  MoveL 7682 to (-24.03, 164.79, 106.87) mm, rotated rx -180 ry 0 rz 180 deg; joints [-52.067, -14.427, 91.412, 80.045, 53.206, -73.667]
  MoveL 7683 to (-24.03, 164.79, 106.87) mm, rotated rx -180 ry 0 rz 180 deg; joints [-52.067, -14.427, 91.412, 80.045, 53.206, -73.667]
  Call Extruder(395.57808)
  MoveL 7684 to (-24.42, 164.75, 106.87) mm, rotated rx 180 ry 0 rz 180 deg; joints [-52.112, -14.466, 91.442, 80.053, 53.25, -73.664]
  MoveL 7685 to (-24.42, 164.75, 106.87) mm, rotated rx 180 ry 0 rz 180 deg; joints [-52.112, -14.466, 91.442, 80.053, 53.25, -73.664]
  Call Extruder(395.77652)
  MoveL 7686 to (-24.8, 164.7, 106.87) mm, rotated rx 180 ry 0 rz 180 deg; joints [-52.156, -14.506, 91.472, 80.062, 53.294, -73.662]
  MoveL 7687 to (-24.8, 164.7, 106.87) mm, rotated rx 180 ry 0 rz 180 deg; joints [-52.156, -14.506, 91.472, 80.062, 53.294, -73.662]
  Call Extruder(395.97583)
  MoveL 7688 to (-25.19, 164.66, 106.87) mm, rotated rx 180 ry 0 rz -180 deg; joints [-52.2, -14.545, 91.501, 80.07, 53.339, -73.659]
  MoveL 7689 to (-25.19, 164.66, 106.87) mm, rotated rx 180 ry 0 rz -180 deg; joints [-52.2, -14.545, 91.501, 80.07, 53.339, -73.659]
  Call Extruder(396.13466)
  MoveL 7690 to (-25.5, 164.61, 106.87) mm, rotated rx 180 ry 0 rz 180 deg; joints [-52.235, -14.578, 91.526, 80.076, 53.373, -73.656]
  MoveL 7691 to (-25.5, 164.61, 106.87) mm, rotated rx 180 ry 0 rz 180 deg; joints [-52.235, -14.578, 91.526, 80.076, 53.373, -73.656]
  Call Extruder(396.29423)
  MoveL 7692 to (-25.8, 164.56, 106.87) mm, rotated rx 180 ry 0 rz 180 deg; joints [-52.269, -14.61, 91.551, 80.082, 53.407, -73.654]
  MoveL 7693 to (-25.8, 164.56, 106.87) mm, rotated rx 180 ry 0 rz 180 deg; joints [-52.269, -14.61, 91.551, 80.082, 53.407, -73.654]
  Call Extruder(396.45451)
  MoveL 7694 to (-26.11, 164.51, 106.87) mm, rotated rx 180 ry 0 rz -180 deg; joints [-52.303, -14.643, 91.575, 80.088, 53.441, -73.651]
  MoveL 7695 to (-26.11, 164.51, 106.87) mm, rotated rx 180 ry 0 rz -180 deg; joints [-52.303, -14.643, 91.575, 80.088, 53.441, -73.651]
  Call Extruder(396.61553)
  MoveL 7696 to (-26.41, 164.46, 106.87) mm, rotated rx -180 ry 0 rz 180 deg; joints [-52.337, -14.675, 91.599, 80.095, 53.475, -73.648]
  MoveL 7697 to (-26.41, 164.46, 106.87) mm, rotated rx -180 ry 0 rz 180 deg; joints [-52.337, -14.675, 91.599, 80.095, 53.475, -73.648]
  Call Extruder(396.77727)
  MoveL 7698 to (-26.72, 164.41, 106.87) mm, rotated rx 180 ry 0 rz 180 deg; joints [-52.371, -14.708, 91.624, 80.101, 53.509, -73.646]
  MoveL 7699 to (-26.72, 164.41, 106.87) mm, rotated rx 180 ry 0 rz 180 deg; joints [-52.371, -14.708, 91.624, 80.101, 53.509, -73.646]
  Call Extruder(396.93974)
  MoveL 7700 to (-27.03, 164.36, 106.87) mm, rotated rx 180 ry 0 rz 180 deg; joints [-52.405, -14.74, 91.648, 80.107, 53.543, -73.643]
  MoveL 7701 to (-27.03, 164.36, 106.87) mm, rotated rx 180 ry 0 rz 180 deg; joints [-52.405, -14.74, 91.648, 80.107, 53.543, -73.643]
  Call Extruder(397.07367)
  MoveL 7702 to (-27.27, 164.32, 106.87) mm, rotated rx 180 ry 0 rz 180 deg; joints [-52.432, -14.768, 91.669, 80.111, 53.57, -73.64]
  MoveL 7703 to (-27.27, 164.32, 106.87) mm, rotated rx 180 ry 0 rz 180 deg; joints [-52.432, -14.768, 91.669, 80.111, 53.57, -73.64]
  Call Extruder(397.20821)
  MoveL 7704 to (-27.52, 164.27, 106.87) mm, rotated rx 180 ry 0 rz 180 deg; joints [-52.459, -14.795, 91.69, 80.116, 53.597, -73.637]
  MoveL 7705 to (-27.52, 164.27, 106.87) mm, rotated rx 180 ry 0 rz 180 deg; joints [-52.459, -14.795, 91.69, 80.116, 53.597, -73.637]
  Call Extruder(397.34335)
  MoveL 7706 to (-27.77, 164.22, 106.87) mm, rotated rx 180 ry 0 rz 180 deg; joints [-52.486, -14.823, 91.71, 80.12, 53.624, -73.634]
  MoveL 7707 to (-27.77, 164.22, 106.87) mm, rotated rx 180 ry 0 rz 180 deg; joints [-52.486, -14.823, 91.71, 80.12, 53.624, -73.634]
  Call Extruder(397.47911)
  MoveL 7708 to (-28.02, 164.17, 106.87) mm, rotated rx 180 ry 0 rz -180 deg; joints [-52.513, -14.85, 91.731, 80.125, 53.651, -73.632]
  MoveL 7709 to (-28.02, 164.17, 106.87) mm, rotated rx 180 ry 0 rz -180 deg; joints [-52.513, -14.85, 91.731, 80.125, 53.651, -73.632]
  Call Extruder(397.61548)
  MoveL 7710 to (-28.27, 164.12, 106.87) mm, rotated rx 180 ry 0 rz 180 deg; joints [-52.54, -14.878, 91.752, 80.129, 53.678, -73.629]
  MoveL 7711 to (-28.27, 164.12, 106.87) mm, rotated rx 180 ry 0 rz 180 deg; joints [-52.54, -14.878, 91.752, 80.129, 53.678, -73.629]
  Call Extruder(397.70034)
  MoveL 7712 to (-28.43, 164.09, 106.87) mm, rotated rx 180 ry 0 rz -180 deg; joints [-52.556, -14.895, 91.764, 80.132, 53.695, -73.627]
  Set speed (130.0 mm/s)
  MoveL 7713 to (-31.76, 163.31, 106.87) mm, rotated rx 180 ry 0 rz 180 deg; joints [-52.91, -15.274, 92.047, 80.186, 54.05, -73.582]
  MoveL 7714 to (-31.76, 163.31, 116.27) mm, rotated rx -180 ry 0 rz 180 deg; joints [-52.91, -15.91, 93.952, 81.097, 53.844, -75.13]
  Call Extruder(395.70034)
  Set speed (40.0 mm/s)
  MoveL 7715 to (-31.76, 163.31, 116.27) mm, rotated rx -180 ry 0 rz 180 deg; joints [-52.91, -15.91, 93.952, 81.097, 53.844, -75.13]
  Call Extruder(0.00000)
  Set speed (130.0 mm/s)
  MoveL 7716 to (-34.23, 161.92, 116.27) mm, rotated rx 180 ry 0 rz 180 deg; joints [-53.095, -16.284, 94.225, 81.084, 54.039, -75.043]
  Call Extruder(2.00000)
  Set speed (40.0 mm/s)
  MoveL 7717 to (-34.23, 161.92, 116.27) mm, rotated rx 180 ry 0 rz 180 deg; joints [-53.095, -16.284, 94.225, 81.084, 54.039, -75.043]
  Set speed (30.0 mm/s)
  MoveL 7718 to (-34.23, 161.92, 116.27) mm, rotated rx 180 ry 0 rz 180 deg; joints [-53.095, -16.284, 94.225, 81.084, 54.039, -75.043]
  Call Extruder(2.16612)
  MoveL 7719 to (-34.45, 161.76, 116.27) mm, rotated rx 180 ry 0 rz 180 deg; joints [-53.109, -16.322, 94.253, 81.081, 54.053, -75.032]
  MoveL 7720 to (-34.45, 161.76, 116.27) mm, rotated rx 180 ry 0 rz 180 deg; joints [-53.109, -16.322, 94.253, 81.081, 54.053, -75.032]
  Call Extruder(2.49954)
  MoveL 7721 to (-34.9, 161.43, 116.27) mm, rotated rx 180 ry 0 rz -180 deg; joints [-53.135, -16.399, 94.309, 81.074, 54.083, -75.012]
  MoveL 7722 to (-34.9, 161.43, 116.27) mm, rotated rx 180 ry 0 rz -180 deg; joints [-53.135, -16.399, 94.309, 81.074, 54.083, -75.012]
  Call Extruder(2.83415)
  MoveL 7723 to (-35.35, 161.1, 116.27) mm, rotated rx 180 ry 0 rz -180 deg; joints [-53.163, -16.476, 94.365, 81.068, 54.112, -74.991]
  Call Extruder(3.66207)
  MoveL 7724 to (-36.39, 160.19, 116.27) mm, rotated rx 180 ry 0 rz 180 deg; joints [-53.209, -16.671, 94.506, 81.044, 54.165, -74.934]
  Call Extruder(4.49000)
  MoveL 7725 to (-37.3, 159.15, 116.27) mm, rotated rx 180 ry 0 rz 180 deg; joints [-53.227, -16.869, 94.649, 81.011, 54.192, -74.87]
  Call Extruder(4.65731)
  MoveL 7726 to (-37.47, 158.93, 116.27) mm, rotated rx 180 ry 0 rz 180 deg; joints [-53.227, -16.909, 94.678, 81.003, 54.193, -74.856]
  MoveL 7727 to (-37.47, 158.93, 116.27) mm, rotated rx 180 ry 0 rz 180 deg; joints [-53.227, -16.909, 94.678, 81.003, 54.193, -74.856]
  Call Extruder(4.99074)
  MoveL 7728 to (-37.8, 158.48, 116.27) mm, rotated rx 180 ry 0 rz -180 deg; joints [-53.226, -16.989, 94.735, 80.986, 54.195, -74.829]
  MoveL 7729 to (-37.8, 158.48, 116.27) mm, rotated rx 180 ry 0 rz -180 deg; joints [-53.226, -16.989, 94.735, 80.986, 54.195, -74.829]
  Call Extruder(5.32299)
  MoveL 7730 to (-38.12, 158.03, 116.27) mm, rotated rx 180 ry 0 rz 180 deg; joints [-53.224, -17.07, 94.793, 80.969, 54.198, -74.801]
  MoveL 7731 to (-38.12, 158.03, 116.27) mm, rotated rx 180 ry 0 rz 180 deg; joints [-53.224, -17.07, 94.793, 80.969, 54.198, -74.801]
  Call Extruder(5.44066)
  MoveL 7732 to (-38.22, 157.85, 116.27) mm, rotated rx 180 ry 0 rz 180 deg; joints [-53.221, -17.098, 94.813, 80.962, 54.195, -74.79]
  MoveL 7733 to (-38.22, 157.85, 116.27) mm, rotated rx 180 ry 0 rz 180 deg; joints [-53.221, -17.098, 94.813, 80.962, 54.195, -74.79]
  Call Extruder(5.64838)
  MoveL 7734 to (-38.4, 157.55, 116.27) mm, rotated rx -180 ry 0 rz 180 deg; joints [-53.214, -17.148, 94.849, 80.95, 54.191, -74.771]
  MoveL 7735 to (-38.4, 157.55, 116.27) mm, rotated rx -180 ry 0 rz 180 deg; joints [-53.214, -17.148, 94.849, 80.95, 54.191, -74.771]
  Call Extruder(5.85533)
  MoveL 7736 to (-38.57, 157.25, 116.27) mm, rotated rx 180 ry 0 rz -180 deg; joints [-53.207, -17.198, 94.885, 80.938, 54.186, -74.753]
  MoveL 7737 to (-38.57, 157.25, 116.27) mm, rotated rx 180 ry 0 rz -180 deg; joints [-53.207, -17.198, 94.885, 80.938, 54.186, -74.753]
  Call Extruder(6.06150)
  MoveL 7738 to (-38.75, 156.94, 116.27) mm, rotated rx -180 ry 0 rz 180 deg; joints [-53.2, -17.248, 94.92, 80.925, 54.182, -74.734]
  MoveL 7739 to (-38.75, 156.94, 116.27) mm, rotated rx -180 ry 0 rz 180 deg; joints [-53.2, -17.248, 94.92, 80.925, 54.182, -74.734]
  Call Extruder(6.24318)
  MoveL 7740 to (-38.89, 156.67, 116.27) mm, rotated rx 180 ry 0 rz 180 deg; joints [-53.191, -17.292, 94.952, 80.913, 54.175, -74.717]
  MoveL 7741 to (-38.89, 156.67, 116.27) mm, rotated rx 180 ry 0 rz 180 deg; joints [-53.191, -17.292, 94.952, 80.913, 54.175, -74.717]
  Call Extruder(6.40116)
  MoveL 7742 to (-39, 156.42, 116.27) mm, rotated rx 180 ry 0 rz 180 deg; joints [-53.18, -17.33, 94.979, 80.902, 54.167, -74.701]
  MoveL 7743 to (-39, 156.42, 116.27) mm, rotated rx 180 ry 0 rz 180 deg; joints [-53.18, -17.33, 94.979, 80.902, 54.167, -74.701]
  Call Extruder(6.55855)
  MoveL 7744 to (-39.11, 156.17, 116.27) mm, rotated rx 180 ry 0 rz 180 deg; joints [-53.17, -17.368, 95.006, 80.891, 54.158, -74.686]
  MoveL 7745 to (-39.11, 156.17, 116.27) mm, rotated rx 180 ry 0 rz 180 deg; joints [-53.17, -17.368, 95.006, 80.891, 54.158, -74.686]
  Call Extruder(6.74127)
  MoveL 7746 to (-39.22, 155.88, 116.27) mm, rotated rx 180 ry 0 rz 180 deg; joints [-53.156, -17.412, 95.037, 80.877, 54.148, -74.668]
  MoveL 7747 to (-39.22, 155.88, 116.27) mm, rotated rx 180 ry 0 rz 180 deg; joints [-53.156, -17.412, 95.037, 80.877, 54.148, -74.668]
  Call Extruder(6.92323)
  MoveL 7748 to (-39.35, 155.58, 116.27) mm, rotated rx 180 ry 0 rz 180 deg; joints [-53.143, -17.456, 95.068, 80.864, 54.137, -74.65]
  MoveL 7749 to (-39.35, 155.58, 116.27) mm, rotated rx 180 ry 0 rz 180 deg; joints [-53.143, -17.456, 95.068, 80.864, 54.137, -74.65]
  Call Extruder(7.07056)
  MoveL 7750 to (-39.44, 155.34, 116.27) mm, rotated rx -180 ry 0 rz 180 deg; joints [-53.131, -17.491, 95.093, 80.853, 54.127, -74.635]
  MoveL 7751 to (-39.44, 155.34, 116.27) mm, rotated rx -180 ry 0 rz 180 deg; joints [-53.131, -17.491, 95.093, 80.853, 54.127, -74.635]
  Call Extruder(7.18380)
  MoveL 7752 to (-39.5, 155.15, 116.27) mm, rotated rx -180 ry 0 rz 180 deg; joints [-53.121, -17.518, 95.112, 80.843, 54.118, -74.623]
  MoveL 7753 to (-39.5, 155.15, 116.27) mm, rotated rx -180 ry 0 rz 180 deg; joints [-53.121, -17.518, 95.112, 80.843, 54.118, -74.623]
  Call Extruder(7.29659)
  MoveL 7754 to (-39.56, 154.97, 116.27) mm, rotated rx 180 ry 0 rz 180 deg; joints [-53.11, -17.545, 95.131, 80.834, 54.109, -74.612]
  MoveL 7755 to (-39.56, 154.97, 116.27) mm, rotated rx 180 ry 0 rz 180 deg; joints [-53.11, -17.545, 95.131, 80.834, 54.109, -74.612]
  Call Extruder(7.40893)
  MoveL 7756 to (-39.62, 154.78, 116.27) mm, rotated rx -180 ry 0 rz 180 deg; joints [-53.099, -17.572, 95.15, 80.825, 54.1, -74.6]
  MoveL 7757 to (-39.62, 154.78, 116.27) mm, rotated rx -180 ry 0 rz 180 deg; joints [-53.099, -17.572, 95.15, 80.825, 54.1, -74.6]
  Call Extruder(7.52083)
  MoveL 7758 to (-39.68, 154.59, 116.27) mm, rotated rx -180 ry 0 rz 180 deg; joints [-53.088, -17.599, 95.169, 80.816, 54.091, -74.588]
  MoveL 7759 to (-39.68, 154.59, 116.27) mm, rotated rx -180 ry 0 rz 180 deg; joints [-53.088, -17.599, 95.169, 80.816, 54.091, -74.588]
  Call Extruder(7.64223)
  MoveL 7760 to (-39.75, 154.38, 116.27) mm, rotated rx 180 ry 0 rz 180 deg; joints [-53.076, -17.628, 95.19, 80.806, 54.08, -74.576]
  MoveL 7761 to (-39.75, 154.38, 116.27) mm, rotated rx 180 ry 0 rz 180 deg; joints [-53.076, -17.628, 95.19, 80.806, 54.08, -74.576]
  Call Extruder(7.77303)
  MoveL 7762 to (-39.81, 154.16, 116.27) mm, rotated rx -180 ry 0 rz 180 deg; joints [-53.063, -17.66, 95.212, 80.795, 54.069, -74.562]
  MoveL 7763 to (-39.81, 154.16, 116.27) mm, rotated rx -180 ry 0 rz 180 deg; joints [-53.063, -17.66, 95.212, 80.795, 54.069, -74.562]
  Call Extruder(7.90326)
  MoveL 7764 to (-39.88, 153.94, 116.27) mm, rotated rx 180 ry 0 rz 180 deg; joints [-53.049, -17.691, 95.234, 80.784, 54.057, -74.548]
  MoveL 7765 to (-39.88, 153.94, 116.27) mm, rotated rx 180 ry 0 rz 180 deg; joints [-53.049, -17.691, 95.234, 80.784, 54.057, -74.548]
  Call Extruder(8.03292)
  MoveL 7766 to (-39.95, 153.71, 116.27) mm, rotated rx 180 ry 0 rz 180 deg; joints [-53.036, -17.723, 95.256, 80.773, 54.046, -74.534]
  MoveL 7767 to (-39.95, 153.71, 116.27) mm, rotated rx 180 ry 0 rz 180 deg; joints [-53.036, -17.723, 95.256, 80.773, 54.046, -74.534]
  Call Extruder(8.16202)
  MoveL 7768 to (-40.02, 153.49, 116.27) mm, rotated rx 180 ry 0 rz 180 deg; joints [-53.022, -17.754, 95.279, 80.761, 54.034, -74.52]
  MoveL 7769 to (-40.02, 153.49, 116.27) mm, rotated rx 180 ry 0 rz 180 deg; joints [-53.022, -17.754, 95.279, 80.761, 54.034, -74.52]
  Call Extruder(8.27711)
  MoveL 7770 to (-40.06, 153.28, 116.27) mm, rotated rx 180 ry 0 rz 180 deg; joints [-53.007, -17.781, 95.298, 80.751, 54.021, -74.507]
  MoveL 7771 to (-40.06, 153.28, 116.27) mm, rotated rx 180 ry 0 rz 180 deg; joints [-53.007, -17.781, 95.298, 80.751, 54.021, -74.507]
  Call Extruder(8.39175)
  MoveL 7772 to (-40.11, 153.08, 116.27) mm, rotated rx 180 ry 0 rz 180 deg; joints [-52.993, -17.809, 95.317, 80.74, 54.008, -74.494]
  MoveL 7773 to (-40.11, 153.08, 116.27) mm, rotated rx 180 ry 0 rz 180 deg; joints [-52.993, -17.809, 95.317, 80.74, 54.008, -74.494]
  Call Extruder(8.50593)
  MoveL 7774 to (-40.15, 152.88, 116.27) mm, rotated rx 180 ry 0 rz 180 deg; joints [-52.978, -17.836, 95.336, 80.729, 53.995, -74.482]
  MoveL 7775 to (-40.15, 152.88, 116.27) mm, rotated rx 180 ry 0 rz 180 deg; joints [-52.978, -17.836, 95.336, 80.729, 53.995, -74.482]
  Call Extruder(8.61966)
  MoveL 7776 to (-40.2, 152.67, 116.27) mm, rotated rx 180 ry 0 rz 180 deg; joints [-52.963, -17.863, 95.355, 80.719, 53.982, -74.469]
  MoveL 7777 to (-40.2, 152.67, 116.27) mm, rotated rx 180 ry 0 rz 180 deg; joints [-52.963, -17.863, 95.355, 80.719, 53.982, -74.469]
  Call Extruder(8.74509)
  MoveL 7778 to (-40.24, 152.44, 116.27) mm, rotated rx -180 ry 0 rz 180 deg; joints [-52.946, -17.893, 95.376, 80.707, 53.968, -74.455]
  MoveL 7779 to (-40.24, 152.44, 116.27) mm, rotated rx -180 ry 0 rz 180 deg; joints [-52.946, -17.893, 95.376, 80.707, 53.968, -74.455]
  Call Extruder(8.88206)
  MoveL 7780 to (-40.29, 152.2, 116.27) mm, rotated rx 180 ry 0 rz 180 deg; joints [-52.928, -17.926, 95.399, 80.694, 53.951, -74.439]
  MoveL 7781 to (-40.29, 152.2, 116.27) mm, rotated rx 180 ry 0 rz 180 deg; joints [-52.928, -17.926, 95.399, 80.694, 53.951, -74.439]
  Call Extruder(9.01843)
  MoveL 7782 to (-40.34, 151.95, 116.27) mm, rotated rx 180 ry 0 rz -180 deg; joints [-52.909, -17.959, 95.422, 80.68, 53.935, -74.423]
  MoveL 7783 to (-40.34, 151.95, 116.27) mm, rotated rx 180 ry 0 rz -180 deg; joints [-52.909, -17.959, 95.422, 80.68, 53.935, -74.423]
  Call Extruder(9.15418)
  MoveL 7784 to (-40.39, 151.7, 116.27) mm, rotated rx 180 ry 0 rz 180 deg; joints [-52.89, -17.991, 95.445, 80.667, 53.918, -74.408]
  MoveL 7785 to (-40.39, 151.7, 116.27) mm, rotated rx 180 ry 0 rz 180 deg; joints [-52.89, -17.991, 95.445, 80.667, 53.918, -74.408]
  Call Extruder(9.28933)
  MoveL 7786 to (-40.44, 151.45, 116.27) mm, rotated rx -180 ry 0 rz 180 deg; joints [-52.871, -18.024, 95.468, 80.654, 53.902, -74.392]
  MoveL 7787 to (-40.44, 151.45, 116.27) mm, rotated rx -180 ry 0 rz 180 deg; joints [-52.871, -18.024, 95.468, 80.654, 53.902, -74.392]
  Call Extruder(9.42386)
  MoveL 7788 to (-40.49, 151.2, 116.27) mm, rotated rx 180 ry 0 rz 180 deg; joints [-52.853, -18.057, 95.491, 80.64, 53.885, -74.376]
  MoveL 7789 to (-40.49, 151.2, 116.27) mm, rotated rx 180 ry 0 rz 180 deg; joints [-52.853, -18.057, 95.491, 80.64, 53.885, -74.376]
  Call Extruder(9.55779)
  MoveL 7790 to (-40.54, 150.95, 116.27) mm, rotated rx 180 ry 0 rz 180 deg; joints [-52.834, -18.09, 95.514, 80.627, 53.869, -74.361]
  MoveL 7791 to (-40.54, 150.95, 116.27) mm, rotated rx 180 ry 0 rz 180 deg; joints [-52.834, -18.09, 95.514, 80.627, 53.869, -74.361]
  Call Extruder(9.70564)
  MoveL 7792 to (-40.59, 150.67, 116.27) mm, rotated rx 180 ry 0 rz 180 deg; joints [-52.812, -18.125, 95.539, 80.612, 53.849, -74.343]
  MoveL 7793 to (-40.59, 150.67, 116.27) mm, rotated rx 180 ry 0 rz 180 deg; joints [-52.812, -18.125, 95.539, 80.612, 53.849, -74.343]
  Call Extruder(9.86737)
  MoveL 7794 to (-40.64, 150.37, 116.27) mm, rotated rx 180 ry 0 rz 180 deg; joints [-52.787, -18.165, 95.566, 80.595, 53.828, -74.324]
  MoveL 7795 to (-40.64, 150.37, 116.27) mm, rotated rx 180 ry 0 rz 180 deg; joints [-52.787, -18.165, 95.566, 80.595, 53.828, -74.324]
  Call Extruder(10.02836)
  MoveL 7796 to (-40.69, 150.06, 116.27) mm, rotated rx 180 ry 0 rz 180 deg; joints [-52.762, -18.204, 95.593, 80.578, 53.805, -74.304]
  MoveL 7797 to (-40.69, 150.06, 116.27) mm, rotated rx 180 ry 0 rz 180 deg; joints [-52.762, -18.204, 95.593, 80.578, 53.805, -74.304]
  Call Extruder(10.18863)
  MoveL 7798 to (-40.73, 149.76, 116.27) mm, rotated rx 180 ry 0 rz 180 deg; joints [-52.737, -18.243, 95.62, 80.561, 53.783, -74.285]
  MoveL 7799 to (-40.73, 149.76, 116.27) mm, rotated rx 180 ry 0 rz 180 deg; joints [-52.737, -18.243, 95.62, 80.561, 53.783, -74.285]
  Call Extruder(10.34817)
  MoveL 7800 to (-40.78, 149.45, 116.27) mm, rotated rx 180 ry 0 rz 180 deg; joints [-52.712, -18.282, 95.648, 80.544, 53.761, -74.265]
  MoveL 7801 to (-40.78, 149.45, 116.27) mm, rotated rx 180 ry 0 rz 180 deg; joints [-52.712, -18.282, 95.648, 80.544, 53.761, -74.265]
  Call Extruder(10.50698)
  MoveL 7802 to (-40.83, 149.14, 116.27) mm, rotated rx 180 ry 0 rz 180 deg; joints [-52.687, -18.321, 95.675, 80.527, 53.739, -74.246]
  MoveL 7803 to (-40.83, 149.14, 116.27) mm, rotated rx 180 ry 0 rz 180 deg; joints [-52.687, -18.321, 95.675, 80.527, 53.739, -74.246]
  Call Extruder(10.68565)
  MoveL 7804 to (-40.88, 148.8, 116.27) mm, rotated rx 180 ry 0 rz 180 deg; joints [-52.658, -18.364, 95.705, 80.508, 53.713, -74.224]
  MoveL 7805 to (-40.88, 148.8, 116.27) mm, rotated rx 180 ry 0 rz 180 deg; joints [-52.658, -18.364, 95.705, 80.508, 53.713, -74.224]
  Call Extruder(10.88409)
  MoveL 7806 to (-40.92, 148.41, 116.27) mm, rotated rx -180 ry 0 rz 180 deg; joints [-52.624, -18.412, 95.738, 80.485, 53.683, -74.199]
  MoveL 7807 to (-40.92, 148.41, 116.27) mm, rotated rx -180 ry 0 rz 180 deg; joints [-52.624, -18.412, 95.738, 80.485, 53.683, -74.199]
  Call Extruder(11.08166)
  MoveL 7808 to (-40.97, 148.02, 116.27) mm, rotated rx 180 ry 0 rz 180 deg; joints [-52.59, -18.46, 95.771, 80.463, 53.653, -74.174]
  MoveL 7809 to (-40.97, 148.02, 116.27) mm, rotated rx 180 ry 0 rz 180 deg; joints [-52.59, -18.46, 95.771, 80.463, 53.653, -74.174]
  Call Extruder(11.27837)
  MoveL 7810 to (-41.02, 147.64, 116.27) mm, rotated rx -180 ry 0 rz -180 deg; joints [-52.556, -18.508, 95.805, 80.441, 53.622, -74.149]
  MoveL 7811 to (-41.02, 147.64, 116.27) mm, rotated rx -180 ry 0 rz -180 deg; joints [-52.556, -18.508, 95.805, 80.441, 53.622, -74.149]
  Call Extruder(11.47421)
  MoveL 7812 to (-41.06, 147.25, 116.27) mm, rotated rx 180 ry 0 rz 180 deg; joints [-52.521, -18.556, 95.838, 80.419, 53.592, -74.124]
  MoveL 7813 to (-41.06, 147.25, 116.27) mm, rotated rx 180 ry 0 rz 180 deg; joints [-52.521, -18.556, 95.838, 80.419, 53.592, -74.124]
  Call Extruder(11.76961)
  MoveL 7814 to (-41.11, 146.66, 116.27) mm, rotated rx 180 ry 0 rz 180 deg; joints [-52.466, -18.627, 95.887, 80.384, 53.542, -74.086]
  MoveL 7815 to (-41.11, 146.66, 116.27) mm, rotated rx 180 ry 0 rz 180 deg; joints [-52.466, -18.627, 95.887, 80.384, 53.542, -74.086]
  Call Extruder(12.06367)
  MoveL 7816 to (-41.15, 146.07, 116.27) mm, rotated rx 180 ry 0 rz 180 deg; joints [-52.411, -18.698, 95.935, 80.349, 53.493, -74.048]
  MoveL 7817 to (-41.15, 146.07, 116.27) mm, rotated rx 180 ry 0 rz 180 deg; joints [-52.411, -18.698, 95.935, 80.349, 53.493, -74.048]
  Call Extruder(12.35641)
  MoveL 7818 to (-41.2, 145.48, 116.27) mm, rotated rx 180 ry 0 rz 180 deg; joints [-52.355, -18.769, 95.984, 80.314, 53.443, -74.009]
  MoveL 7819 to (-41.2, 145.48, 116.27) mm, rotated rx 180 ry 0 rz 180 deg; joints [-52.355, -18.769, 95.984, 80.314, 53.443, -74.009]
  Call Extruder(12.92986)
  MoveL 7820 to (-41.25, 144.32, 116.27) mm, rotated rx 180 ry 0 rz 180 deg; joints [-52.239, -18.904, 96.077, 80.242, 53.338, -73.933]
  MoveL 7821 to (-41.25, 144.32, 116.27) mm, rotated rx 180 ry 0 rz 180 deg; joints [-52.239, -18.904, 96.077, 80.242, 53.338, -73.933]
  Call Extruder(13.64382)
  MoveL 7822 to (-41.29, 142.86, 116.27) mm, rotated rx 180 ry 0 rz 180 deg; joints [-52.09, -19.071, 96.191, 80.152, 53.204, -73.837]
  Call Extruder(55.70865)
  MoveL 7823 to (-41.29, 57.14, 116.27) mm, rotated rx -180 ry 0 rz 180 deg; joints [-40.759, -27.817, 101.5, 71.946, 43.368, -65.849]
  Call Extruder(56.13720)
  MoveL 7824 to (-41.27, 56.26, 116.27) mm, rotated rx 180 ry 0 rz -180 deg; joints [-40.614, -27.893, 101.541, 71.824, 43.248, -65.737]
  MoveL 7825 to (-41.27, 56.26, 116.27) mm, rotated rx 180 ry 0 rz -180 deg; joints [-40.614, -27.893, 101.541, 71.824, 43.248, -65.737]
  Call Extruder(56.71065)
  MoveL 7826 to (-41.23, 55.1, 116.27) mm, rotated rx 180 ry 0 rz -180 deg; joints [-40.419, -27.992, 101.593, 71.659, 43.084, -65.586]
  MoveL 7827 to (-41.23, 55.1, 116.27) mm, rotated rx 180 ry 0 rz -180 deg; joints [-40.419, -27.992, 101.593, 71.659, 43.084, -65.586]
  Call Extruder(57.14497)
  MoveL 7828 to (-41.18, 54.23, 116.27) mm, rotated rx -180 ry 0 rz 180 deg; joints [-40.269, -28.066, 101.632, 71.533, 42.958, -65.471]
  MoveL 7829 to (-41.18, 54.23, 116.27) mm, rotated rx -180 ry 0 rz 180 deg; joints [-40.269, -28.066, 101.632, 71.533, 42.958, -65.471]
  Call Extruder(57.43904)
  MoveL 7830 to (-41.13, 53.64, 116.27) mm, rotated rx 180 ry 0 rz 180 deg; joints [-40.165, -28.113, 101.657, 71.446, 42.871, -65.394]
  MoveL 7831 to (-41.13, 53.64, 116.27) mm, rotated rx 180 ry 0 rz 180 deg; joints [-40.165, -28.113, 101.657, 71.446, 42.871, -65.394]
  Call Extruder(57.73444)
  MoveL 7832 to (-41.09, 53.05, 116.27) mm, rotated rx 180 ry 0 rz 180 deg; joints [-40.062, -28.16, 101.681, 71.36, 42.784, -65.316]
  MoveL 7833 to (-41.09, 53.05, 116.27) mm, rotated rx 180 ry 0 rz 180 deg; joints [-40.062, -28.16, 101.681, 71.36, 42.784, -65.316]
  Call Extruder(57.98067)
  MoveL 7834 to (-41.04, 52.56, 116.27) mm, rotated rx 180 ry 0 rz 180 deg; joints [-39.975, -28.198, 101.702, 71.288, 42.711, -65.251]
  MoveL 7835 to (-41.04, 52.56, 116.27) mm, rotated rx 180 ry 0 rz 180 deg; joints [-39.975, -28.198, 101.702, 71.288, 42.711, -65.251]
  Call Extruder(58.17738)
  MoveL 7836 to (-40.99, 52.17, 116.27) mm, rotated rx 180 ry 0 rz 180 deg; joints [-39.904, -28.228, 101.717, 71.23, 42.652, -65.2]
  MoveL 7837 to (-40.99, 52.17, 116.27) mm, rotated rx 180 ry 0 rz 180 deg; joints [-39.904, -28.228, 101.717, 71.23, 42.652, -65.2]
  Call Extruder(58.37495)
  MoveL 7838 to (-40.95, 51.78, 116.27) mm, rotated rx -180 ry 0 rz -180 deg; joints [-39.833, -28.257, 101.732, 71.172, 42.592, -65.148]
  MoveL 7839 to (-40.95, 51.78, 116.27) mm, rotated rx -180 ry 0 rz -180 deg; joints [-39.833, -28.257, 101.732, 71.172, 42.592, -65.148]
  Call Extruder(58.57339)
  MoveL 7840 to (-40.9, 51.4, 116.27) mm, rotated rx 180 ry 0 rz 180 deg; joints [-39.763, -28.286, 101.748, 71.113, 42.532, -65.096]
  MoveL 7841 to (-40.9, 51.4, 116.27) mm, rotated rx 180 ry 0 rz 180 deg; joints [-39.763, -28.286, 101.748, 71.113, 42.532, -65.096]
  Call Extruder(58.77270)
  MoveL 7842 to (-40.86, 51.01, 116.27) mm, rotated rx 180 ry 0 rz 180 deg; joints [-39.692, -28.315, 101.763, 71.055, 42.472, -65.044]
  MoveL 7843 to (-40.86, 51.01, 116.27) mm, rotated rx 180 ry 0 rz 180 deg; joints [-39.692, -28.315, 101.763, 71.055, 42.472, -65.044]
  Call Extruder(58.93152)
  MoveL 7844 to (-40.81, 50.7, 116.27) mm, rotated rx 180 ry 0 rz -180 deg; joints [-39.634, -28.337, 101.774, 71.008, 42.423, -65.003]
  MoveL 7845 to (-40.81, 50.7, 116.27) mm, rotated rx 180 ry 0 rz -180 deg; joints [-39.634, -28.337, 101.774, 71.008, 42.423, -65.003]
  Call Extruder(59.09106)
  MoveL 7846 to (-40.76, 50.4, 116.27) mm, rotated rx 180 ry 0 rz -180 deg; joints [-39.576, -28.359, 101.785, 70.961, 42.374, -64.962]
  MoveL 7847 to (-40.76, 50.4, 116.27) mm, rotated rx 180 ry 0 rz -180 deg; joints [-39.576, -28.359, 101.785, 70.961, 42.374, -64.962]
  Call Extruder(59.25133)
  MoveL 7848 to (-40.71, 50.09, 116.27) mm, rotated rx 180 ry 0 rz 180 deg; joints [-39.518, -28.38, 101.797, 70.914, 42.325, -64.92]
  MoveL 7849 to (-40.71, 50.09, 116.27) mm, rotated rx 180 ry 0 rz 180 deg; joints [-39.518, -28.38, 101.797, 70.914, 42.325, -64.92]
  Call Extruder(59.41232)
  MoveL 7850 to (-40.66, 49.79, 116.27) mm, rotated rx -180 ry 0 rz 180 deg; joints [-39.46, -28.402, 101.808, 70.867, 42.276, -64.879]
  MoveL 7851 to (-40.66, 49.79, 116.27) mm, rotated rx -180 ry 0 rz 180 deg; joints [-39.46, -28.402, 101.808, 70.867, 42.276, -64.879]
  Call Extruder(59.57405)
  MoveL 7852 to (-40.61, 49.48, 116.27) mm, rotated rx 180 ry 0 rz 180 deg; joints [-39.402, -28.423, 101.819, 70.819, 42.227, -64.837]
  MoveL 7853 to (-40.61, 49.48, 116.27) mm, rotated rx 180 ry 0 rz 180 deg; joints [-39.402, -28.423, 101.819, 70.819, 42.227, -64.837]
  Call Extruder(59.73650)
  MoveL 7854 to (-40.57, 49.17, 116.27) mm, rotated rx 180 ry 0 rz 180 deg; joints [-39.344, -28.445, 101.83, 70.772, 42.178, -64.796]
  MoveL 7855 to (-40.57, 49.17, 116.27) mm, rotated rx 180 ry 0 rz 180 deg; joints [-39.344, -28.445, 101.83, 70.772, 42.178, -64.796]
  Call Extruder(59.87043)
  MoveL 7856 to (-40.52, 48.93, 116.27) mm, rotated rx 180 ry 0 rz -180 deg; joints [-39.296, -28.461, 101.839, 70.733, 42.137, -64.761]
  MoveL 7857 to (-40.52, 48.93, 116.27) mm, rotated rx 180 ry 0 rz -180 deg; joints [-39.296, -28.461, 101.839, 70.733, 42.137, -64.761]
  Call Extruder(60.00496)
  MoveL 7858 to (-40.47, 48.68, 116.27) mm, rotated rx 180 ry 0 rz 180 deg; joints [-39.247, -28.477, 101.847, 70.693, 42.095, -64.727]
  MoveL 7859 to (-40.47, 48.68, 116.27) mm, rotated rx 180 ry 0 rz 180 deg; joints [-39.247, -28.477, 101.847, 70.693, 42.095, -64.727]
  Call Extruder(60.14011)
  MoveL 7860 to (-40.42, 48.43, 116.27) mm, rotated rx 180 ry 0 rz 180 deg; joints [-39.198, -28.494, 101.856, 70.654, 42.053, -64.693]
  MoveL 7861 to (-40.42, 48.43, 116.27) mm, rotated rx 180 ry 0 rz 180 deg; joints [-39.198, -28.494, 101.856, 70.654, 42.053, -64.693]
  Call Extruder(60.27586)
  MoveL 7862 to (-40.37, 48.18, 116.27) mm, rotated rx -180 ry 0 rz -180 deg; joints [-39.149, -28.51, 101.864, 70.615, 42.012, -64.659]
  MoveL 7863 to (-40.37, 48.18, 116.27) mm, rotated rx -180 ry 0 rz -180 deg; joints [-39.149, -28.51, 101.864, 70.615, 42.012, -64.659]
  Call Extruder(60.41223)
  MoveL 7864 to (-40.32, 47.93, 116.27) mm, rotated rx 180 ry 0 rz 180 deg; joints [-39.1, -28.526, 101.873, 70.575, 41.97, -64.625]
  MoveL 7865 to (-40.32, 47.93, 116.27) mm, rotated rx 180 ry 0 rz 180 deg; joints [-39.1, -28.526, 101.873, 70.575, 41.97, -64.625]
  Call Extruder(60.54920)
  MoveL 7866 to (-40.27, 47.68, 116.27) mm, rotated rx 180 ry 0 rz 180 deg; joints [-39.051, -28.543, 101.881, 70.536, 41.929, -64.59]
  MoveL 7867 to (-40.27, 47.68, 116.27) mm, rotated rx 180 ry 0 rz 180 deg; joints [-39.051, -28.543, 101.881, 70.536, 41.929, -64.59]
  Call Extruder(60.68679)
  MoveL 7868 to (-40.22, 47.43, 116.27) mm, rotated rx 180 ry 0 rz -180 deg; joints [-39.002, -28.559, 101.889, 70.496, 41.887, -64.556]
  MoveL 7869 to (-40.22, 47.43, 116.27) mm, rotated rx 180 ry 0 rz -180 deg; joints [-39.002, -28.559, 101.889, 70.496, 41.887, -64.556]
  Call Extruder(60.80052)
  MoveL 7870 to (-40.17, 47.23, 116.27) mm, rotated rx 180 ry 0 rz 180 deg; joints [-38.962, -28.572, 101.896, 70.463, 41.852, -64.528]
  MoveL 7871 to (-40.17, 47.23, 116.27) mm, rotated rx 180 ry 0 rz 180 deg; joints [-38.962, -28.572, 101.896, 70.463, 41.852, -64.528]
  Call Extruder(60.91470)
  MoveL 7872 to (-40.13, 47.02, 116.27) mm, rotated rx 180 ry 0 rz 180 deg; joints [-38.921, -28.585, 101.903, 70.43, 41.817, -64.499]
  MoveL 7873 to (-40.13, 47.02, 116.27) mm, rotated rx 180 ry 0 rz 180 deg; joints [-38.921, -28.585, 101.903, 70.43, 41.817, -64.499]
  Call Extruder(61.02933)
  MoveL 7874 to (-40.08, 46.82, 116.27) mm, rotated rx 180 ry 0 rz -180 deg; joints [-38.88, -28.597, 101.909, 70.397, 41.783, -64.471]
  MoveL 7875 to (-40.08, 46.82, 116.27) mm, rotated rx 180 ry 0 rz -180 deg; joints [-38.88, -28.597, 101.909, 70.397, 41.783, -64.471]
  Call Extruder(61.14442)
  MoveL 7876 to (-40.04, 46.61, 116.27) mm, rotated rx 180 ry 0 rz -180 deg; joints [-38.839, -28.61, 101.916, 70.364, 41.748, -64.442]
  MoveL 7877 to (-40.04, 46.61, 116.27) mm, rotated rx 180 ry 0 rz -180 deg; joints [-38.839, -28.61, 101.916, 70.364, 41.748, -64.442]
  Call Extruder(61.26666)
  MoveL 7878 to (-39.98, 46.4, 116.27) mm, rotated rx 180 ry 0 rz 180 deg; joints [-38.795, -28.623, 101.922, 70.33, 41.71, -64.413]
  MoveL 7879 to (-39.98, 46.4, 116.27) mm, rotated rx 180 ry 0 rz 180 deg; joints [-38.795, -28.623, 101.922, 70.33, 41.71, -64.413]
  Call Extruder(61.39632)
  MoveL 7880 to (-39.92, 46.18, 116.27) mm, rotated rx 180 ry 0 rz 180 deg; joints [-38.748, -28.634, 101.929, 70.293, 41.669, -64.381]
  MoveL 7881 to (-39.92, 46.18, 116.27) mm, rotated rx 180 ry 0 rz 180 deg; joints [-38.748, -28.634, 101.929, 70.293, 41.669, -64.381]
  Call Extruder(61.52655)
  MoveL 7882 to (-39.85, 45.95, 116.27) mm, rotated rx 180 ry 0 rz 180 deg; joints [-38.7, -28.646, 101.935, 70.256, 41.629, -64.35]
  MoveL 7883 to (-39.85, 45.95, 116.27) mm, rotated rx 180 ry 0 rz 180 deg; joints [-38.7, -28.646, 101.935, 70.256, 41.629, -64.35]
  Call Extruder(61.65735)
  MoveL 7884 to (-39.78, 45.73, 116.27) mm, rotated rx 180 ry 0 rz 180 deg; joints [-38.653, -28.658, 101.941, 70.219, 41.588, -64.319]
  MoveL 7885 to (-39.78, 45.73, 116.27) mm, rotated rx 180 ry 0 rz 180 deg; joints [-38.653, -28.658, 101.941, 70.219, 41.588, -64.319]
  Call Extruder(61.78871)
  MoveL 7886 to (-39.71, 45.5, 116.27) mm, rotated rx 180 ry 0 rz 180 deg; joints [-38.605, -28.67, 101.947, 70.181, 41.547, -64.287]
  MoveL 7887 to (-39.71, 45.5, 116.27) mm, rotated rx 180 ry 0 rz 180 deg; joints [-38.605, -28.67, 101.947, 70.181, 41.547, -64.287]
  Call Extruder(61.90061)
  MoveL 7888 to (-39.65, 45.32, 116.27) mm, rotated rx -180 ry 0 rz 180 deg; joints [-38.565, -28.68, 101.952, 70.15, 41.512, -64.261]
  MoveL 7889 to (-39.65, 45.32, 116.27) mm, rotated rx -180 ry 0 rz 180 deg; joints [-38.565, -28.68, 101.952, 70.15, 41.512, -64.261]
  Call Extruder(62.01295)
  MoveL 7890 to (-39.59, 45.13, 116.27) mm, rotated rx 180 ry 0 rz 180 deg; joints [-38.524, -28.689, 101.957, 70.118, 41.477, -64.235]
  MoveL 7891 to (-39.59, 45.13, 116.27) mm, rotated rx 180 ry 0 rz 180 deg; joints [-38.524, -28.689, 101.957, 70.118, 41.477, -64.235]
  Call Extruder(62.12574)
  MoveL 7892 to (-39.53, 44.94, 116.27) mm, rotated rx 180 ry 0 rz 180 deg; joints [-38.483, -28.699, 101.962, 70.087, 41.442, -64.208]
  MoveL 7893 to (-39.53, 44.94, 116.27) mm, rotated rx 180 ry 0 rz 180 deg; joints [-38.483, -28.699, 101.962, 70.087, 41.442, -64.208]
  Call Extruder(62.23898)
  MoveL 7894 to (-39.47, 44.75, 116.27) mm, rotated rx 180 ry 0 rz 180 deg; joints [-38.443, -28.708, 101.967, 70.055, 41.407, -64.181]
  MoveL 7895 to (-39.47, 44.75, 116.27) mm, rotated rx 180 ry 0 rz 180 deg; joints [-38.443, -28.708, 101.967, 70.055, 41.407, -64.181]
  Call Extruder(62.35266)
  MoveL 7896 to (-39.41, 44.56, 116.27) mm, rotated rx 180 ry 0 rz 180 deg; joints [-38.402, -28.718, 101.972, 70.024, 41.372, -64.155]
  MoveL 7897 to (-39.41, 44.56, 116.27) mm, rotated rx 180 ry 0 rz 180 deg; joints [-38.402, -28.718, 101.972, 70.024, 41.372, -64.155]
  Call Extruder(62.53462)
  MoveL 7898 to (-39.29, 44.27, 116.27) mm, rotated rx -180 ry 0 rz -180 deg; joints [-38.335, -28.73, 101.978, 69.973, 41.314, -64.114]
  MoveL 7899 to (-39.29, 44.27, 116.27) mm, rotated rx -180 ry 0 rz -180 deg; joints [-38.335, -28.73, 101.978, 69.973, 41.314, -64.114]
  Call Extruder(62.71734)
  MoveL 7900 to (-39.16, 43.98, 116.27) mm, rotated rx 180 ry 0 rz 180 deg; joints [-38.269, -28.741, 101.984, 69.923, 41.256, -64.072]
  MoveL 7901 to (-39.16, 43.98, 116.27) mm, rotated rx 180 ry 0 rz 180 deg; joints [-38.269, -28.741, 101.984, 69.923, 41.256, -64.072]
  Call Extruder(62.88775)
  MoveL 7902 to (-39.05, 43.71, 116.27) mm, rotated rx -180 ry 0 rz 180 deg; joints [-38.207, -28.752, 101.989, 69.876, 41.202, -64.034]
  MoveL 7903 to (-39.05, 43.71, 116.27) mm, rotated rx -180 ry 0 rz 180 deg; joints [-38.207, -28.752, 101.989, 69.876, 41.202, -64.034]
  Call Extruder(63.04573)
  MoveL 7904 to (-38.94, 43.46, 116.27) mm, rotated rx 180 ry 0 rz 180 deg; joints [-38.149, -28.761, 101.994, 69.833, 41.152, -63.999]
  MoveL 7905 to (-38.94, 43.46, 116.27) mm, rotated rx 180 ry 0 rz 180 deg; joints [-38.149, -28.761, 101.994, 69.833, 41.152, -63.999]
  Call Extruder(63.20432)
  MoveL 7906 to (-38.84, 43.21, 116.27) mm, rotated rx 180 ry 0 rz 180 deg; joints [-38.092, -28.771, 101.999, 69.79, 41.102, -63.963]
  MoveL 7907 to (-38.84, 43.21, 116.27) mm, rotated rx 180 ry 0 rz 180 deg; joints [-38.092, -28.771, 101.999, 69.79, 41.102, -63.963]
  Call Extruder(63.41049)
  MoveL 7908 to (-38.66, 42.91, 116.27) mm, rotated rx 180 ry 0 rz 180 deg; joints [-38.016, -28.778, 102.003, 69.735, 41.034, -63.92]
  MoveL 7909 to (-38.66, 42.91, 116.27) mm, rotated rx 180 ry 0 rz 180 deg; joints [-38.016, -28.778, 102.003, 69.735, 41.034, -63.92]
  Call Extruder(63.61743)
  MoveL 7910 to (-38.49, 42.6, 116.27) mm, rotated rx -180 ry 0 rz 180 deg; joints [-37.939, -28.785, 102.006, 69.681, 40.967, -63.877]
  MoveL 7911 to (-38.49, 42.6, 116.27) mm, rotated rx -180 ry 0 rz 180 deg; joints [-37.939, -28.785, 102.006, 69.681, 40.967, -63.877]
  Call Extruder(63.82516)
  MoveL 7912 to (-38.31, 42.3, 116.27) mm, rotated rx 180 ry 0 rz 180 deg; joints [-37.863, -28.791, 102.009, 69.626, 40.9, -63.833]
  MoveL 7913 to (-38.31, 42.3, 116.27) mm, rotated rx 180 ry 0 rz 180 deg; joints [-37.863, -28.791, 102.009, 69.626, 40.9, -63.833]
  Call Extruder(64.03366)
  MoveL 7914 to (-38.14, 41.99, 116.27) mm, rotated rx -180 ry 0 rz 180 deg; joints [-37.787, -28.798, 102.013, 69.571, 40.832, -63.79]
  MoveL 7915 to (-38.14, 41.99, 116.27) mm, rotated rx -180 ry 0 rz 180 deg; joints [-37.787, -28.798, 102.013, 69.571, 40.832, -63.79]
  Call Extruder(64.21320)
  MoveL 7916 to (-37.96, 41.75, 116.27) mm, rotated rx -180 ry 0 rz 180 deg; joints [-37.72, -28.799, 102.013, 69.525, 40.773, -63.755]
  MoveL 7917 to (-37.96, 41.75, 116.27) mm, rotated rx -180 ry 0 rz 180 deg; joints [-37.72, -28.799, 102.013, 69.525, 40.773, -63.755]
  Call Extruder(64.54664)
  MoveL 7918 to (-37.63, 41.3, 116.27) mm, rotated rx 180 ry 0 rz 180 deg; joints [-37.598, -28.801, 102.015, 69.441, 40.664, -63.69]
  MoveL 7919 to (-37.63, 41.3, 116.27) mm, rotated rx 180 ry 0 rz 180 deg; joints [-37.598, -28.801, 102.015, 69.441, 40.664, -63.69]
  Call Extruder(64.88126)
  MoveL 7920 to (-37.3, 40.85, 116.27) mm, rotated rx 180 ry 0 rz 180 deg; joints [-37.475, -28.803, 102.016, 69.356, 40.554, -63.625]
  Call Extruder(65.70919)
  MoveL 7921 to (-36.39, 39.81, 116.27) mm, rotated rx 180 ry 0 rz 180 deg; joints [-37.173, -28.79, 102.009, 69.156, 40.281, -63.477]
  Call Extruder(66.53710)
  MoveL 7922 to (-35.35, 38.9, 116.27) mm, rotated rx 180 ry 0 rz 180 deg; joints [-36.876, -28.752, 101.989, 68.97, 40.009, -63.346]
  Call Extruder(66.70441)
  MoveL 7923 to (-35.13, 38.73, 116.27) mm, rotated rx 180 ry 0 rz -180 deg; joints [-36.818, -28.741, 101.983, 68.935, 39.955, -63.323]
  MoveL 7924 to (-35.13, 38.73, 116.27) mm, rotated rx 180 ry 0 rz -180 deg; joints [-36.818, -28.741, 101.983, 68.935, 39.955, -63.323]
  Call Extruder(67.03783)
  MoveL 7925 to (-34.68, 38.41, 116.27) mm, rotated rx 180 ry 0 rz -180 deg; joints [-36.701, -28.718, 101.972, 68.866, 39.846, -63.276]
  MoveL 7926 to (-34.68, 38.41, 116.27) mm, rotated rx 180 ry 0 rz -180 deg; joints [-36.701, -28.718, 101.972, 68.866, 39.846, -63.276]
  Call Extruder(67.37007)
  MoveL 7927 to (-34.22, 38.08, 116.27) mm, rotated rx 180 ry 0 rz 180 deg; joints [-36.584, -28.695, 101.96, 68.796, 39.738, -63.229]
  MoveL 7928 to (-34.22, 38.08, 116.27) mm, rotated rx 180 ry 0 rz 180 deg; joints [-36.584, -28.695, 101.96, 68.796, 39.738, -63.229]
  Call Extruder(67.48778)
  MoveL 7929 to (-34.05, 37.98, 116.27) mm, rotated rx 180 ry 0 rz -180 deg; joints [-36.544, -28.685, 101.954, 68.774, 39.701, -63.215]
  MoveL 7930 to (-34.05, 37.98, 116.27) mm, rotated rx 180 ry 0 rz -180 deg; joints [-36.544, -28.685, 101.954, 68.774, 39.701, -63.215]
  Call Extruder(67.69550)
  MoveL 7931 to (-33.75, 37.8, 116.27) mm, rotated rx 180 ry 0 rz -180 deg; joints [-36.474, -28.666, 101.945, 68.734, 39.634, -63.19]
  MoveL 7932 to (-33.75, 37.8, 116.27) mm, rotated rx 180 ry 0 rz -180 deg; joints [-36.474, -28.666, 101.945, 68.734, 39.634, -63.19]
  Call Extruder(67.90244)
  MoveL 7933 to (-33.45, 37.63, 116.27) mm, rotated rx 180 ry 0 rz 180 deg; joints [-36.403, -28.646, 101.935, 68.695, 39.568, -63.165]
  MoveL 7934 to (-33.45, 37.63, 116.27) mm, rotated rx 180 ry 0 rz 180 deg; joints [-36.403, -28.646, 101.935, 68.695, 39.568, -63.165]
  Call Extruder(68.10860)
  MoveL 7935 to (-33.14, 37.45, 116.27) mm, rotated rx 180 ry 0 rz 180 deg; joints [-36.333, -28.627, 101.925, 68.656, 39.502, -63.14]
  MoveL 7936 to (-33.14, 37.45, 116.27) mm, rotated rx 180 ry 0 rz 180 deg; joints [-36.333, -28.627, 101.925, 68.656, 39.502, -63.14]
  Call Extruder(68.29029)
  MoveL 7937 to (-32.86, 37.31, 116.27) mm, rotated rx 180 ry 0 rz 180 deg; joints [-36.272, -28.608, 101.915, 68.623, 39.445, -63.12]
  MoveL 7938 to (-32.86, 37.31, 116.27) mm, rotated rx 180 ry 0 rz 180 deg; joints [-36.272, -28.608, 101.915, 68.623, 39.445, -63.12]
  Call Extruder(68.44829)
  MoveL 7939 to (-32.62, 37.2, 116.27) mm, rotated rx 180 ry 0 rz 180 deg; joints [-36.221, -28.589, 101.905, 68.597, 39.396, -63.106]
  MoveL 7940 to (-32.62, 37.2, 116.27) mm, rotated rx 180 ry 0 rz 180 deg; joints [-36.221, -28.589, 101.905, 68.597, 39.396, -63.106]
  Call Extruder(68.60569)
  MoveL 7941 to (-32.37, 37.09, 116.27) mm, rotated rx -180 ry 0 rz 180 deg; joints [-36.17, -28.57, 101.895, 68.571, 39.347, -63.091]
  MoveL 7942 to (-32.37, 37.09, 116.27) mm, rotated rx -180 ry 0 rz 180 deg; joints [-36.17, -28.57, 101.895, 68.571, 39.347, -63.091]
  Call Extruder(68.78840)
  MoveL 7943 to (-32.08, 36.97, 116.27) mm, rotated rx 180 ry 0 rz 180 deg; joints [-36.112, -28.548, 101.884, 68.541, 39.291, -63.075]
  MoveL 7944 to (-32.08, 36.97, 116.27) mm, rotated rx 180 ry 0 rz 180 deg; joints [-36.112, -28.548, 101.884, 68.541, 39.291, -63.075]
  Call Extruder(68.97035)
  MoveL 7945 to (-31.78, 36.85, 116.27) mm, rotated rx -180 ry 0 rz 180 deg; joints [-36.053, -28.525, 101.872, 68.512, 39.234, -63.058]
  MoveL 7946 to (-31.78, 36.85, 116.27) mm, rotated rx -180 ry 0 rz 180 deg; joints [-36.053, -28.525, 101.872, 68.512, 39.234, -63.058]
  Call Extruder(69.11768)
  MoveL 7947 to (-31.54, 36.76, 116.27) mm, rotated rx 180 ry 0 rz 180 deg; joints [-36.006, -28.506, 101.862, 68.489, 39.189, -63.046]
  MoveL 7948 to (-31.54, 36.76, 116.27) mm, rotated rx 180 ry 0 rz 180 deg; joints [-36.006, -28.506, 101.862, 68.489, 39.189, -63.046]
  Call Extruder(69.23091)
  MoveL 7949 to (-31.35, 36.7, 116.27) mm, rotated rx -180 ry 0 rz 180 deg; joints [-35.971, -28.49, 101.854, 68.472, 39.155, -63.037]
  MoveL 7950 to (-31.35, 36.7, 116.27) mm, rotated rx -180 ry 0 rz 180 deg; joints [-35.971, -28.49, 101.854, 68.472, 39.155, -63.037]
  Call Extruder(69.34371)
  MoveL 7951 to (-31.17, 36.64, 116.27) mm, rotated rx 180 ry 0 rz 180 deg; joints [-35.936, -28.474, 101.845, 68.456, 39.121, -63.029]
  MoveL 7952 to (-31.17, 36.64, 116.27) mm, rotated rx 180 ry 0 rz 180 deg; joints [-35.936, -28.474, 101.845, 68.456, 39.121, -63.029]
  Call Extruder(69.45605)
  MoveL 7953 to (-30.98, 36.58, 116.27) mm, rotated rx 180 ry 0 rz -180 deg; joints [-35.901, -28.458, 101.837, 68.44, 39.087, -63.021]
  MoveL 7954 to (-30.98, 36.58, 116.27) mm, rotated rx 180 ry 0 rz -180 deg; joints [-35.901, -28.458, 101.837, 68.44, 39.087, -63.021]
  Call Extruder(69.56796)
  MoveL 7955 to (-30.79, 36.52, 116.27) mm, rotated rx 180 ry 0 rz 180 deg; joints [-35.867, -28.442, 101.829, 68.424, 39.054, -63.013]
  MoveL 7956 to (-30.79, 36.52, 116.27) mm, rotated rx 180 ry 0 rz 180 deg; joints [-35.867, -28.442, 101.829, 68.424, 39.054, -63.013]
  Call Extruder(69.68936)
  MoveL 7957 to (-30.58, 36.45, 116.27) mm, rotated rx 180 ry 0 rz 180 deg; joints [-35.829, -28.424, 101.819, 68.406, 39.017, -63.005]
  MoveL 7958 to (-30.58, 36.45, 116.27) mm, rotated rx 180 ry 0 rz 180 deg; joints [-35.829, -28.424, 101.819, 68.406, 39.017, -63.005]
  Call Extruder(69.82015)
  MoveL 7959 to (-30.36, 36.38, 116.27) mm, rotated rx -180 ry 0 rz 180 deg; joints [-35.788, -28.405, 101.809, 68.388, 38.978, -62.996]
  MoveL 7960 to (-30.36, 36.38, 116.27) mm, rotated rx -180 ry 0 rz 180 deg; joints [-35.788, -28.405, 101.809, 68.388, 38.978, -62.996]
  Call Extruder(69.95037)
  MoveL 7961 to (-30.14, 36.32, 116.27) mm, rotated rx 180 ry 0 rz 180 deg; joints [-35.748, -28.385, 101.799, 68.369, 38.938, -62.987]
  MoveL 7962 to (-30.14, 36.32, 116.27) mm, rotated rx 180 ry 0 rz 180 deg; joints [-35.748, -28.385, 101.799, 68.369, 38.938, -62.987]
  Call Extruder(70.08003)
  MoveL 7963 to (-29.91, 36.25, 116.27) mm, rotated rx 180 ry 0 rz 180 deg; joints [-35.708, -28.366, 101.789, 68.351, 38.899, -62.978]
  MoveL 7964 to (-29.91, 36.25, 116.27) mm, rotated rx 180 ry 0 rz 180 deg; joints [-35.708, -28.366, 101.789, 68.351, 38.899, -62.978]
  Call Extruder(70.20913)
  MoveL 7965 to (-29.69, 36.18, 116.27) mm, rotated rx 180 ry 0 rz 180 deg; joints [-35.668, -28.346, 101.779, 68.333, 38.86, -62.969]
  MoveL 7966 to (-29.69, 36.18, 116.27) mm, rotated rx 180 ry 0 rz 180 deg; joints [-35.668, -28.346, 101.779, 68.333, 38.86, -62.969]
  Call Extruder(70.32420)
  MoveL 7967 to (-29.48, 36.14, 116.27) mm, rotated rx 180 ry 0 rz -180 deg; joints [-35.634, -28.327, 101.769, 68.319, 38.826, -62.964]
  MoveL 7968 to (-29.48, 36.14, 116.27) mm, rotated rx 180 ry 0 rz -180 deg; joints [-35.634, -28.327, 101.769, 68.319, 38.826, -62.964]
  Call Extruder(70.43882)
  MoveL 7969 to (-29.28, 36.09, 116.27) mm, rotated rx 180 ry 0 rz 180 deg; joints [-35.601, -28.308, 101.759, 68.305, 38.793, -62.958]
  MoveL 7970 to (-29.28, 36.09, 116.27) mm, rotated rx 180 ry 0 rz 180 deg; joints [-35.601, -28.308, 101.759, 68.305, 38.793, -62.958]
  Call Extruder(70.55299)
  MoveL 7971 to (-29.08, 36.05, 116.27) mm, rotated rx 180 ry 0 rz 180 deg; joints [-35.567, -28.288, 101.749, 68.291, 38.76, -62.953]
  MoveL 7972 to (-29.08, 36.05, 116.27) mm, rotated rx 180 ry 0 rz 180 deg; joints [-35.567, -28.288, 101.749, 68.291, 38.76, -62.953]
  Call Extruder(70.66671)
  MoveL 7973 to (-28.87, 36, 116.27) mm, rotated rx -180 ry 0 rz 180 deg; joints [-35.533, -28.269, 101.739, 68.278, 38.726, -62.948]
  MoveL 7974 to (-28.87, 36, 116.27) mm, rotated rx -180 ry 0 rz 180 deg; joints [-35.533, -28.269, 101.739, 68.278, 38.726, -62.948]
  Call Extruder(70.79213)
  MoveL 7975 to (-28.64, 35.96, 116.27) mm, rotated rx 180 ry 0 rz 180 deg; joints [-35.497, -28.248, 101.727, 68.263, 38.69, -62.942]
  MoveL 7976 to (-28.64, 35.96, 116.27) mm, rotated rx 180 ry 0 rz 180 deg; joints [-35.497, -28.248, 101.727, 68.263, 38.69, -62.942]
  Call Extruder(70.92911)
  MoveL 7977 to (-28.4, 35.91, 116.27) mm, rotated rx 180 ry 0 rz 180 deg; joints [-35.457, -28.224, 101.715, 68.247, 38.65, -62.936]
  MoveL 7978 to (-28.4, 35.91, 116.27) mm, rotated rx 180 ry 0 rz 180 deg; joints [-35.457, -28.224, 101.715, 68.247, 38.65, -62.936]
  Call Extruder(71.06547)
  MoveL 7979 to (-28.15, 35.86, 116.27) mm, rotated rx 180 ry 0 rz 180 deg; joints [-35.417, -28.2, 101.702, 68.231, 38.61, -62.93]
  MoveL 7980 to (-28.15, 35.86, 116.27) mm, rotated rx 180 ry 0 rz 180 deg; joints [-35.417, -28.2, 101.702, 68.231, 38.61, -62.93]
  Call Extruder(71.20123)
  MoveL 7981 to (-27.9, 35.81, 116.27) mm, rotated rx 180 ry 0 rz 180 deg; joints [-35.377, -28.176, 101.69, 68.215, 38.57, -62.924]
  MoveL 7982 to (-27.9, 35.81, 116.27) mm, rotated rx 180 ry 0 rz 180 deg; joints [-35.377, -28.176, 101.69, 68.215, 38.57, -62.924]
  Call Extruder(71.33638)
  MoveL 7983 to (-27.65, 35.76, 116.27) mm, rotated rx 180 ry 0 rz 180 deg; joints [-35.337, -28.152, 101.677, 68.199, 38.531, -62.919]
  MoveL 7984 to (-27.65, 35.76, 116.27) mm, rotated rx 180 ry 0 rz 180 deg; joints [-35.337, -28.152, 101.677, 68.199, 38.531, -62.919]
  Call Extruder(71.47091)
  MoveL 7985 to (-27.4, 35.71, 116.27) mm, rotated rx -180 ry 0 rz 180 deg; joints [-35.297, -28.128, 101.665, 68.183, 38.491, -62.913]
  MoveL 7986 to (-27.4, 35.71, 116.27) mm, rotated rx -180 ry 0 rz 180 deg; joints [-35.297, -28.128, 101.665, 68.183, 38.491, -62.913]
  Call Extruder(71.60484)
  MoveL 7987 to (-27.15, 35.66, 116.27) mm, rotated rx 180 ry 0 rz 180 deg; joints [-35.258, -28.104, 101.652, 68.168, 38.452, -62.907]
  MoveL 7988 to (-27.15, 35.66, 116.27) mm, rotated rx 180 ry 0 rz 180 deg; joints [-35.258, -28.104, 101.652, 68.168, 38.452, -62.907]
  Call Extruder(71.75270)
  MoveL 7989 to (-26.87, 35.61, 116.27) mm, rotated rx 180 ry 0 rz 180 deg; joints [-35.215, -28.077, 101.638, 68.151, 38.409, -62.902]
  MoveL 7990 to (-26.87, 35.61, 116.27) mm, rotated rx 180 ry 0 rz 180 deg; joints [-35.215, -28.077, 101.638, 68.151, 38.409, -62.902]
  Call Extruder(71.91443)
  MoveL 7991 to (-26.57, 35.56, 116.27) mm, rotated rx 180 ry 0 rz 180 deg; joints [-35.168, -28.046, 101.621, 68.134, 38.362, -62.896]
  MoveL 7992 to (-26.57, 35.56, 116.27) mm, rotated rx 180 ry 0 rz 180 deg; joints [-35.168, -28.046, 101.621, 68.134, 38.362, -62.896]
  Call Extruder(72.07544)
  MoveL 7993 to (-26.26, 35.51, 116.27) mm, rotated rx 180 ry 0 rz 180 deg; joints [-35.122, -28.016, 101.605, 68.117, 38.315, -62.891]
  MoveL 7994 to (-26.26, 35.51, 116.27) mm, rotated rx 180 ry 0 rz 180 deg; joints [-35.122, -28.016, 101.605, 68.117, 38.315, -62.891]
  Call Extruder(72.23572)
  MoveL 7995 to (-25.96, 35.47, 116.27) mm, rotated rx 180 ry 0 rz 180 deg; joints [-35.075, -27.985, 101.589, 68.1, 38.269, -62.886]
  MoveL 7996 to (-25.96, 35.47, 116.27) mm, rotated rx 180 ry 0 rz 180 deg; joints [-35.075, -27.985, 101.589, 68.1, 38.269, -62.886]
  Call Extruder(72.39527)
  MoveL 7997 to (-25.65, 35.42, 116.27) mm, rotated rx 180 ry 0 rz 180 deg; joints [-35.029, -27.955, 101.573, 68.083, 38.222, -62.881]
  MoveL 7998 to (-25.65, 35.42, 116.27) mm, rotated rx 180 ry 0 rz 180 deg; joints [-35.029, -27.955, 101.573, 68.083, 38.222, -62.881]
  Call Extruder(72.55409)
  MoveL 7999 to (-25.34, 35.37, 116.27) mm, rotated rx -180 ry 0 rz 180 deg; joints [-34.983, -27.924, 101.557, 68.066, 38.176, -62.876]
  MoveL 8000 to (-25.34, 35.37, 116.27) mm, rotated rx -180 ry 0 rz 180 deg; joints [-34.983, -27.924, 101.557, 68.066, 38.176, -62.876]
  Call Extruder(72.73276)
  MoveL 8001 to (-25, 35.32, 116.27) mm, rotated rx -180 ry 0 rz 180 deg; joints [-34.932, -27.889, 101.538, 68.048, 38.124, -62.871]
  MoveL 8002 to (-25, 35.32, 116.27) mm, rotated rx -180 ry 0 rz 180 deg; joints [-34.932, -27.889, 101.538, 68.048, 38.124, -62.871]
  Call Extruder(72.93120)
  MoveL 8003 to (-24.61, 35.28, 116.27) mm, rotated rx 180 ry 0 rz 180 deg; joints [-34.877, -27.849, 101.517, 68.029, 38.068, -62.867]
  MoveL 8004 to (-24.61, 35.28, 116.27) mm, rotated rx 180 ry 0 rz 180 deg; joints [-34.877, -27.849, 101.517, 68.029, 38.068, -62.867]
  Call Extruder(73.12878)
  MoveL 8005 to (-24.22, 35.23, 116.27) mm, rotated rx -180 ry 0 rz 180 deg; joints [-34.821, -27.809, 101.496, 68.01, 38.011, -62.863]
  MoveL 8006 to (-24.22, 35.23, 116.27) mm, rotated rx -180 ry 0 rz 180 deg; joints [-34.821, -27.809, 101.496, 68.01, 38.011, -62.863]
  Call Extruder(73.32549)
  MoveL 8007 to (-23.83, 35.18, 116.27) mm, rotated rx 180 ry 0 rz 180 deg; joints [-34.766, -27.768, 101.474, 67.992, 37.955, -62.859]
  MoveL 8008 to (-23.83, 35.18, 116.27) mm, rotated rx 180 ry 0 rz 180 deg; joints [-34.766, -27.768, 101.474, 67.992, 37.955, -62.859]
  Call Extruder(73.52132)
  MoveL 8009 to (-23.45, 35.14, 116.27) mm, rotated rx 180 ry 0 rz 180 deg; joints [-34.711, -27.728, 101.453, 67.973, 37.899, -62.856]
  MoveL 8010 to (-23.45, 35.14, 116.27) mm, rotated rx 180 ry 0 rz 180 deg; joints [-34.711, -27.728, 101.453, 67.973, 37.899, -62.856]
  Call Extruder(73.81672)
  MoveL 8011 to (-22.86, 35.09, 116.27) mm, rotated rx -180 ry 0 rz 180 deg; joints [-34.631, -27.665, 101.419, 67.949, 37.817, -62.853]
  MoveL 8012 to (-22.86, 35.09, 116.27) mm, rotated rx -180 ry 0 rz 180 deg; joints [-34.631, -27.665, 101.419, 67.949, 37.817, -62.853]
  Call Extruder(74.11078)
  MoveL 8013 to (-22.27, 35.04, 116.27) mm, rotated rx -180 ry 0 rz -180 deg; joints [-34.552, -27.602, 101.385, 67.925, 37.736, -62.851]
  MoveL 8014 to (-22.27, 35.04, 116.27) mm, rotated rx -180 ry 0 rz -180 deg; joints [-34.552, -27.602, 101.385, 67.925, 37.736, -62.851]
  Call Extruder(74.40351)
  MoveL 8015 to (-21.68, 35, 116.27) mm, rotated rx 180 ry 0 rz 180 deg; joints [-34.473, -27.539, 101.352, 67.901, 37.654, -62.849]
  MoveL 8016 to (-21.68, 35, 116.27) mm, rotated rx 180 ry 0 rz 180 deg; joints [-34.473, -27.539, 101.352, 67.901, 37.654, -62.849]
  Call Extruder(74.97696)
  MoveL 8017 to (-20.52, 34.95, 116.27) mm, rotated rx 180 ry 0 rz 180 deg; joints [-34.326, -27.41, 101.283, 67.863, 37.501, -62.852]
  MoveL 8018 to (-20.52, 34.95, 116.27) mm, rotated rx 180 ry 0 rz 180 deg; joints [-34.326, -27.41, 101.283, 67.863, 37.501, -62.852]
  Call Extruder(75.69093)
  MoveL 8019 to (-19.06, 34.91, 116.27) mm, rotated rx 180 ry 0 rz 180 deg; joints [-34.146, -27.247, 101.195, 67.819, 37.313, -62.859]
  Call Extruder(192.53767)
  MoveL 8020 to (219.06, 34.91, 116.27) mm, rotated rx 180 ry 0 rz 180 deg; joints [-18.248, 4.688, 75.276, 62.142, 20.743, -60.526]
  Call Extruder(192.96623)
  MoveL 8021 to (219.94, 34.93, 116.27) mm, rotated rx 180 ry 0 rz 180 deg; joints [-18.218, 4.824, 75.129, 62.075, 20.722, -60.46]
  MoveL 8022 to (219.94, 34.93, 116.27) mm, rotated rx 180 ry 0 rz 180 deg; joints [-18.218, 4.824, 75.129, 62.075, 20.722, -60.46]
  Call Extruder(193.53967)
  MoveL 8023 to (221.1, 34.98, 116.27) mm, rotated rx 180 ry 0 rz 180 deg; joints [-18.181, 5.007, 74.931, 61.988, 20.697, -60.374]
  MoveL 8024 to (221.1, 34.98, 116.27) mm, rotated rx 180 ry 0 rz 180 deg; joints [-18.181, 5.007, 74.931, 61.988, 20.697, -60.374]
  Call Extruder(193.97399)
  MoveL 8025 to (221.97, 35.02, 116.27) mm, rotated rx 180 ry 0 rz -180 deg; joints [-18.154, 5.145, 74.781, 61.923, 20.679, -60.309]
  MoveL 8026 to (221.97, 35.02, 116.27) mm, rotated rx 180 ry 0 rz -180 deg; joints [-18.154, 5.145, 74.781, 61.923, 20.679, -60.309]
  Call Extruder(194.26805)
  MoveL 8027 to (222.56, 35.07, 116.27) mm, rotated rx 180 ry 0 rz 180 deg; joints [-18.138, 5.239, 74.679, 61.881, 20.669, -60.268]
  MoveL 8028 to (222.56, 35.07, 116.27) mm, rotated rx 180 ry 0 rz 180 deg; joints [-18.138, 5.239, 74.679, 61.881, 20.669, -60.268]
  Call Extruder(194.56344)
  MoveL 8029 to (223.15, 35.11, 116.27) mm, rotated rx 180 ry 0 rz 180 deg; joints [-18.121, 5.334, 74.576, 61.839, 20.658, -60.226]
  MoveL 8030 to (223.15, 35.11, 116.27) mm, rotated rx 180 ry 0 rz 180 deg; joints [-18.121, 5.334, 74.576, 61.839, 20.658, -60.226]
  Call Extruder(194.80967)
  MoveL 8031 to (223.64, 35.16, 116.27) mm, rotated rx 180 ry 0 rz 180 deg; joints [-18.109, 5.412, 74.491, 61.805, 20.651, -60.192]
  MoveL 8032 to (223.64, 35.16, 116.27) mm, rotated rx 180 ry 0 rz 180 deg; joints [-18.109, 5.412, 74.491, 61.805, 20.651, -60.192]
  Call Extruder(195.00638)
  MoveL 8033 to (224.03, 35.21, 116.27) mm, rotated rx 180 ry 0 rz 180 deg; joints [-18.1, 5.475, 74.422, 61.779, 20.646, -60.166]
  MoveL 8034 to (224.03, 35.21, 116.27) mm, rotated rx 180 ry 0 rz 180 deg; joints [-18.1, 5.475, 74.422, 61.779, 20.646, -60.166]
  Call Extruder(195.20395)
  MoveL 8035 to (224.42, 35.25, 116.27) mm, rotated rx 180 ry 0 rz 180 deg; joints [-18.091, 5.538, 74.354, 61.753, 20.641, -60.139]
  MoveL 8036 to (224.42, 35.25, 116.27) mm, rotated rx 180 ry 0 rz 180 deg; joints [-18.091, 5.538, 74.354, 61.753, 20.641, -60.139]
  Call Extruder(195.40240)
  MoveL 8037 to (224.8, 35.3, 116.27) mm, rotated rx -180 ry 0 rz -180 deg; joints [-18.082, 5.601, 74.285, 61.727, 20.636, -60.113]
  MoveL 8038 to (224.8, 35.3, 116.27) mm, rotated rx -180 ry 0 rz -180 deg; joints [-18.082, 5.601, 74.285, 61.727, 20.636, -60.113]
  Call Extruder(195.60171)
  MoveL 8039 to (225.19, 35.34, 116.27) mm, rotated rx 180 ry 0 rz 180 deg; joints [-18.073, 5.664, 74.216, 61.7, 20.631, -60.087]
  MoveL 8040 to (225.19, 35.34, 116.27) mm, rotated rx 180 ry 0 rz 180 deg; joints [-18.073, 5.664, 74.216, 61.7, 20.631, -60.087]
  Call Extruder(195.76053)
  MoveL 8041 to (225.5, 35.39, 116.27) mm, rotated rx 180 ry 0 rz 180 deg; joints [-18.068, 5.714, 74.161, 61.681, 20.628, -60.067]
  MoveL 8042 to (225.5, 35.39, 116.27) mm, rotated rx 180 ry 0 rz 180 deg; joints [-18.068, 5.714, 74.161, 61.681, 20.628, -60.067]
  Call Extruder(195.92007)
  MoveL 8043 to (225.8, 35.44, 116.27) mm, rotated rx -180 ry 0 rz 180 deg; joints [-18.062, 5.764, 74.106, 61.662, 20.626, -60.048]
  MoveL 8044 to (225.8, 35.44, 116.27) mm, rotated rx -180 ry 0 rz 180 deg; joints [-18.062, 5.764, 74.106, 61.662, 20.626, -60.048]
  Call Extruder(196.08035)
  MoveL 8045 to (226.11, 35.49, 116.27) mm, rotated rx 180 ry 0 rz 180 deg; joints [-18.056, 5.815, 74.051, 61.643, 20.623, -60.028]
  MoveL 8046 to (226.11, 35.49, 116.27) mm, rotated rx 180 ry 0 rz 180 deg; joints [-18.056, 5.815, 74.051, 61.643, 20.623, -60.028]
  Call Extruder(196.24135)
  MoveL 8047 to (226.41, 35.54, 116.27) mm, rotated rx 180 ry 0 rz 180 deg; joints [-18.051, 5.865, 73.996, 61.623, 20.62, -60.009]
  MoveL 8048 to (226.41, 35.54, 116.27) mm, rotated rx 180 ry 0 rz 180 deg; joints [-18.051, 5.865, 73.996, 61.623, 20.62, -60.009]
  Call Extruder(196.40308)
  MoveL 8049 to (226.72, 35.59, 116.27) mm, rotated rx -180 ry 0 rz 180 deg; joints [-18.045, 5.915, 73.94, 61.604, 20.618, -59.989]
  MoveL 8050 to (226.72, 35.59, 116.27) mm, rotated rx -180 ry 0 rz 180 deg; joints [-18.045, 5.915, 73.94, 61.604, 20.618, -59.989]
  Call Extruder(196.56554)
  MoveL 8051 to (227.03, 35.63, 116.27) mm, rotated rx -180 ry 0 rz 180 deg; joints [-18.039, 5.966, 73.885, 61.584, 20.615, -59.969]
  MoveL 8052 to (227.03, 35.63, 116.27) mm, rotated rx -180 ry 0 rz 180 deg; joints [-18.039, 5.966, 73.885, 61.584, 20.615, -59.969]
  Call Extruder(196.69947)
  MoveL 8053 to (227.27, 35.68, 116.27) mm, rotated rx 180 ry 0 rz 180 deg; joints [-18.036, 6.008, 73.839, 61.569, 20.614, -59.954]
  MoveL 8054 to (227.27, 35.68, 116.27) mm, rotated rx 180 ry 0 rz 180 deg; joints [-18.036, 6.008, 73.839, 61.569, 20.614, -59.954]
  Call Extruder(196.83401)
  MoveL 8055 to (227.52, 35.73, 116.27) mm, rotated rx 180 ry 0 rz 180 deg; joints [-18.033, 6.049, 73.793, 61.555, 20.613, -59.939]
  MoveL 8056 to (227.52, 35.73, 116.27) mm, rotated rx 180 ry 0 rz 180 deg; joints [-18.033, 6.049, 73.793, 61.555, 20.613, -59.939]
  Call Extruder(196.96915)
  MoveL 8057 to (227.77, 35.78, 116.27) mm, rotated rx 180 ry 0 rz 180 deg; joints [-18.029, 6.091, 73.747, 61.54, 20.612, -59.924]
  MoveL 8058 to (227.77, 35.78, 116.27) mm, rotated rx 180 ry 0 rz 180 deg; joints [-18.029, 6.091, 73.747, 61.54, 20.612, -59.924]
  Call Extruder(197.10491)
  MoveL 8059 to (228.02, 35.83, 116.27) mm, rotated rx 180 ry 0 rz 180 deg; joints [-18.026, 6.133, 73.701, 61.525, 20.611, -59.909]
  MoveL 8060 to (228.02, 35.83, 116.27) mm, rotated rx 180 ry 0 rz 180 deg; joints [-18.026, 6.133, 73.701, 61.525, 20.611, -59.909]
  Call Extruder(197.24128)
  MoveL 8061 to (228.27, 35.88, 116.27) mm, rotated rx 180 ry 0 rz 180 deg; joints [-18.022, 6.174, 73.655, 61.51, 20.61, -59.893]
  MoveL 8062 to (228.27, 35.88, 116.27) mm, rotated rx 180 ry 0 rz 180 deg; joints [-18.022, 6.174, 73.655, 61.51, 20.61, -59.893]
  Call Extruder(197.37826)
  MoveL 8063 to (228.52, 35.93, 116.27) mm, rotated rx 180 ry 0 rz 180 deg; joints [-18.019, 6.216, 73.61, 61.495, 20.61, -59.878]
  MoveL 8064 to (228.52, 35.93, 116.27) mm, rotated rx 180 ry 0 rz 180 deg; joints [-18.019, 6.216, 73.61, 61.495, 20.61, -59.878]
  Call Extruder(197.51585)
  MoveL 8065 to (228.77, 35.98, 116.27) mm, rotated rx 180 ry 0 rz 180 deg; joints [-18.015, 6.258, 73.563, 61.48, 20.609, -59.863]
  MoveL 8066 to (228.77, 35.98, 116.27) mm, rotated rx 180 ry 0 rz 180 deg; joints [-18.015, 6.258, 73.563, 61.48, 20.609, -59.863]
  Call Extruder(197.62957)
  MoveL 8067 to (228.97, 36.03, 116.27) mm, rotated rx 180 ry 0 rz 180 deg; joints [-18.013, 6.292, 73.526, 61.468, 20.608, -59.85]
  MoveL 8068 to (228.97, 36.03, 116.27) mm, rotated rx 180 ry 0 rz 180 deg; joints [-18.013, 6.292, 73.526, 61.468, 20.608, -59.85]
  Call Extruder(197.74374)
  MoveL 8069 to (229.18, 36.07, 116.27) mm, rotated rx 180 ry 0 rz -180 deg; joints [-18.01, 6.327, 73.487, 61.457, 20.608, -59.838]
  MoveL 8070 to (229.18, 36.07, 116.27) mm, rotated rx 180 ry 0 rz -180 deg; joints [-18.01, 6.327, 73.487, 61.457, 20.608, -59.838]
  Call Extruder(197.85836)
  MoveL 8071 to (229.38, 36.12, 116.27) mm, rotated rx 180 ry 0 rz 180 deg; joints [-18.008, 6.361, 73.449, 61.445, 20.608, -59.826]
  MoveL 8072 to (229.38, 36.12, 116.27) mm, rotated rx 180 ry 0 rz 180 deg; joints [-18.008, 6.361, 73.449, 61.445, 20.608, -59.826]
  Call Extruder(197.97344)
  MoveL 8073 to (229.59, 36.16, 116.27) mm, rotated rx 180 ry 0 rz -180 deg; joints [-18.006, 6.395, 73.411, 61.433, 20.607, -59.814]
  MoveL 8074 to (229.59, 36.16, 116.27) mm, rotated rx 180 ry 0 rz -180 deg; joints [-18.006, 6.395, 73.411, 61.433, 20.607, -59.814]
  Call Extruder(198.09430)
  MoveL 8075 to (229.8, 36.21, 116.27) mm, rotated rx -180 ry 0 rz 180 deg; joints [-18.004, 6.432, 73.371, 61.421, 20.608, -59.802]
  MoveL 8076 to (229.8, 36.21, 116.27) mm, rotated rx -180 ry 0 rz 180 deg; joints [-18.004, 6.432, 73.371, 61.421, 20.608, -59.802]
  Call Extruder(198.22115)
  MoveL 8077 to (230.02, 36.28, 116.27) mm, rotated rx 180 ry 0 rz 180 deg; joints [-18.003, 6.47, 73.329, 61.411, 20.609, -59.791]
  MoveL 8078 to (230.02, 36.28, 116.27) mm, rotated rx 180 ry 0 rz 180 deg; joints [-18.003, 6.47, 73.329, 61.411, 20.609, -59.791]
  Call Extruder(198.33995)
  MoveL 8079 to (230.22, 36.34, 116.27) mm, rotated rx 180 ry 0 rz 180 deg; joints [-18.003, 6.505, 73.29, 61.401, 20.61, -59.78]
  MoveL 8080 to (230.22, 36.34, 116.27) mm, rotated rx 180 ry 0 rz 180 deg; joints [-18.003, 6.505, 73.29, 61.401, 20.61, -59.78]
  Call Extruder(198.45066)
  MoveL 8081 to (230.41, 36.4, 116.27) mm, rotated rx 180 ry 0 rz 180 deg; joints [-18.002, 6.538, 73.254, 61.392, 20.612, -59.771]
  MoveL 8082 to (230.41, 36.4, 116.27) mm, rotated rx 180 ry 0 rz 180 deg; joints [-18.002, 6.538, 73.254, 61.392, 20.612, -59.771]
  Call Extruder(198.56179)
  MoveL 8083 to (230.6, 36.46, 116.27) mm, rotated rx 180 ry 0 rz 180 deg; joints [-18.002, 6.571, 73.217, 61.384, 20.613, -59.762]
  MoveL 8084 to (230.6, 36.46, 116.27) mm, rotated rx 180 ry 0 rz 180 deg; joints [-18.002, 6.571, 73.217, 61.384, 20.613, -59.762]
  Call Extruder(198.67341)
  MoveL 8085 to (230.79, 36.52, 116.27) mm, rotated rx -180 ry 0 rz 180 deg; joints [-18.002, 6.604, 73.181, 61.375, 20.615, -59.753]
  MoveL 8086 to (230.79, 36.52, 116.27) mm, rotated rx -180 ry 0 rz 180 deg; joints [-18.002, 6.604, 73.181, 61.375, 20.615, -59.753]
  Call Extruder(198.78553)
  MoveL 8087 to (230.98, 36.58, 116.27) mm, rotated rx 180 ry 0 rz 180 deg; joints [-18.002, 6.636, 73.144, 61.367, 20.617, -59.744]
  MoveL 8088 to (230.98, 36.58, 116.27) mm, rotated rx 180 ry 0 rz 180 deg; joints [-18.002, 6.636, 73.144, 61.367, 20.617, -59.744]
  Call Extruder(198.89810)
  MoveL 8089 to (231.17, 36.64, 116.27) mm, rotated rx -180 ry 0 rz 180 deg; joints [-18.002, 6.669, 73.107, 61.358, 20.618, -59.735]
  MoveL 8090 to (231.17, 36.64, 116.27) mm, rotated rx -180 ry 0 rz 180 deg; joints [-18.002, 6.669, 73.107, 61.358, 20.618, -59.735]
  Call Extruder(199.01111)
  MoveL 8091 to (231.35, 36.7, 116.27) mm, rotated rx 180 ry 0 rz -180 deg; joints [-18.002, 6.702, 73.071, 61.35, 20.62, -59.726]
  MoveL 8092 to (231.35, 36.7, 116.27) mm, rotated rx 180 ry 0 rz -180 deg; joints [-18.002, 6.702, 73.071, 61.35, 20.62, -59.726]
  Call Extruder(199.12456)
  MoveL 8093 to (231.54, 36.76, 116.27) mm, rotated rx 180 ry 0 rz 180 deg; joints [-18.002, 6.735, 73.034, 61.341, 20.622, -59.716]
  MoveL 8094 to (231.54, 36.76, 116.27) mm, rotated rx 180 ry 0 rz 180 deg; joints [-18.002, 6.735, 73.034, 61.341, 20.622, -59.716]
  Call Extruder(199.27220)
  MoveL 8095 to (231.78, 36.85, 116.27) mm, rotated rx -180 ry 0 rz 180 deg; joints [-18.004, 6.778, 72.987, 61.332, 20.625, -59.706]
  MoveL 8096 to (231.78, 36.85, 116.27) mm, rotated rx -180 ry 0 rz 180 deg; joints [-18.004, 6.778, 72.987, 61.332, 20.625, -59.706]
  Call Extruder(199.45454)
  MoveL 8097 to (232.07, 36.98, 116.27) mm, rotated rx 180 ry 0 rz 180 deg; joints [-18.006, 6.83, 72.928, 61.322, 20.631, -59.695]
  MoveL 8098 to (232.07, 36.98, 116.27) mm, rotated rx 180 ry 0 rz 180 deg; joints [-18.006, 6.83, 72.928, 61.322, 20.631, -59.695]
  Call Extruder(199.63764)
  MoveL 8099 to (232.37, 37.09, 116.27) mm, rotated rx 180 ry 0 rz 180 deg; joints [-18.009, 6.883, 72.87, 61.312, 20.636, -59.684]
  MoveL 8100 to (232.37, 37.09, 116.27) mm, rotated rx 180 ry 0 rz 180 deg; joints [-18.009, 6.883, 72.87, 61.312, 20.636, -59.684]
  Call Extruder(199.79534)
  MoveL 8101 to (232.62, 37.2, 116.27) mm, rotated rx 180 ry 0 rz 180 deg; joints [-18.012, 6.928, 72.82, 61.304, 20.641, -59.675]
  MoveL 8102 to (232.62, 37.2, 116.27) mm, rotated rx 180 ry 0 rz 180 deg; joints [-18.012, 6.928, 72.82, 61.304, 20.641, -59.675]
  Call Extruder(199.95364)
  MoveL 8103 to (232.87, 37.31, 116.27) mm, rotated rx 180 ry 0 rz -180 deg; joints [-18.015, 6.973, 72.77, 61.296, 20.646, -59.666]
  MoveL 8104 to (232.87, 37.31, 116.27) mm, rotated rx 180 ry 0 rz -180 deg; joints [-18.015, 6.973, 72.77, 61.296, 20.646, -59.666]
  Call Extruder(200.13566)
  MoveL 8105 to (233.14, 37.45, 116.27) mm, rotated rx 180 ry 0 rz 180 deg; joints [-18.02, 7.024, 72.712, 61.29, 20.654, -59.659]
  MoveL 8106 to (233.14, 37.45, 116.27) mm, rotated rx 180 ry 0 rz 180 deg; joints [-18.02, 7.024, 72.712, 61.29, 20.654, -59.659]
  Call Extruder(200.34222)
  MoveL 8107 to (233.45, 37.63, 116.27) mm, rotated rx -180 ry 0 rz 180 deg; joints [-18.029, 7.081, 72.648, 61.287, 20.664, -59.653]
  MoveL 8108 to (233.45, 37.63, 116.27) mm, rotated rx -180 ry 0 rz 180 deg; joints [-18.029, 7.081, 72.648, 61.287, 20.664, -59.653]
  Call Extruder(200.54955)
  MoveL 8109 to (233.75, 37.8, 116.27) mm, rotated rx 180 ry 0 rz 180 deg; joints [-18.037, 7.139, 72.584, 61.283, 20.674, -59.647]
  MoveL 8110 to (233.75, 37.8, 116.27) mm, rotated rx 180 ry 0 rz 180 deg; joints [-18.037, 7.139, 72.584, 61.283, 20.674, -59.647]
  Call Extruder(200.75767)
  MoveL 8111 to (234.05, 37.98, 116.27) mm, rotated rx -180 ry 0 rz 180 deg; joints [-18.045, 7.196, 72.52, 61.279, 20.685, -59.642]
  MoveL 8112 to (234.05, 37.98, 116.27) mm, rotated rx -180 ry 0 rz 180 deg; joints [-18.045, 7.196, 72.52, 61.279, 20.685, -59.642]
  Call Extruder(200.87539)
  MoveL 8113 to (234.23, 38.08, 116.27) mm, rotated rx 180 ry 0 rz 180 deg; joints [-18.05, 7.228, 72.484, 61.276, 20.691, -59.638]
  MoveL 8114 to (234.23, 38.08, 116.27) mm, rotated rx 180 ry 0 rz 180 deg; joints [-18.05, 7.228, 72.484, 61.276, 20.691, -59.638]
  Call Extruder(201.20821)
  MoveL 8115 to (234.68, 38.41, 116.27) mm, rotated rx 180 ry 0 rz 180 deg; joints [-18.07, 7.317, 72.384, 61.28, 20.713, -59.638]
  MoveL 8116 to (234.68, 38.41, 116.27) mm, rotated rx 180 ry 0 rz 180 deg; joints [-18.07, 7.317, 72.384, 61.28, 20.713, -59.638]
  Call Extruder(201.54222)
  MoveL 8117 to (235.13, 38.73, 116.27) mm, rotated rx 180 ry 0 rz -180 deg; joints [-18.089, 7.406, 72.285, 61.282, 20.735, -59.637]
  MoveL 8118 to (235.13, 38.73, 116.27) mm, rotated rx 180 ry 0 rz -180 deg; joints [-18.089, 7.406, 72.285, 61.282, 20.735, -59.637]
  Call Extruder(201.70980)
  MoveL 8119 to (235.35, 38.9, 116.27) mm, rotated rx 180 ry 0 rz -180 deg; joints [-18.099, 7.451, 72.235, 61.284, 20.746, -59.636]
  Call Extruder(202.53913)
  MoveL 8120 to (236.39, 39.81, 116.27) mm, rotated rx -180 ry 0 rz -180 deg; joints [-18.16, 7.663, 71.995, 61.31, 20.812, -59.652]
  Call Extruder(203.17020)
  MoveL 8121 to (237.09, 40.59, 116.27) mm, rotated rx -180 ry 0 rz 180 deg; joints [-18.22, 7.816, 71.823, 61.349, 20.873, -59.683]
  MoveL 8122 to (237.09, 40.59, 116.27) mm, rotated rx -180 ry 0 rz 180 deg; joints [-18.22, 7.816, 71.823, 61.349, 20.873, -59.683]
  Call Extruder(203.36780)
  MoveL 8123 to (237.3, 40.85, 116.27) mm, rotated rx -180 ry 0 rz 180 deg; joints [-18.24, 7.864, 71.769, 61.363, 20.893, -59.694]
  Call Extruder(203.70181)
  MoveL 8124 to (237.63, 41.3, 116.27) mm, rotated rx 180 ry 0 rz 180 deg; joints [-18.277, 7.94, 71.683, 61.392, 20.929, -59.718]
  MoveL 8125 to (237.63, 41.3, 116.27) mm, rotated rx 180 ry 0 rz 180 deg; joints [-18.277, 7.94, 71.683, 61.392, 20.929, -59.718]
  Call Extruder(204.03463)
  MoveL 8126 to (237.96, 41.75, 116.27) mm, rotated rx 180 ry 0 rz -180 deg; joints [-18.313, 8.016, 71.596, 61.42, 20.966, -59.741]
  MoveL 8127 to (237.96, 41.75, 116.27) mm, rotated rx 180 ry 0 rz -180 deg; joints [-18.313, 8.016, 71.596, 61.42, 20.966, -59.741]
  Call Extruder(204.21387)
  MoveL 8128 to (238.13, 41.99, 116.27) mm, rotated rx 180 ry 0 rz 180 deg; joints [-18.333, 8.057, 71.55, 61.436, 20.986, -59.754]
